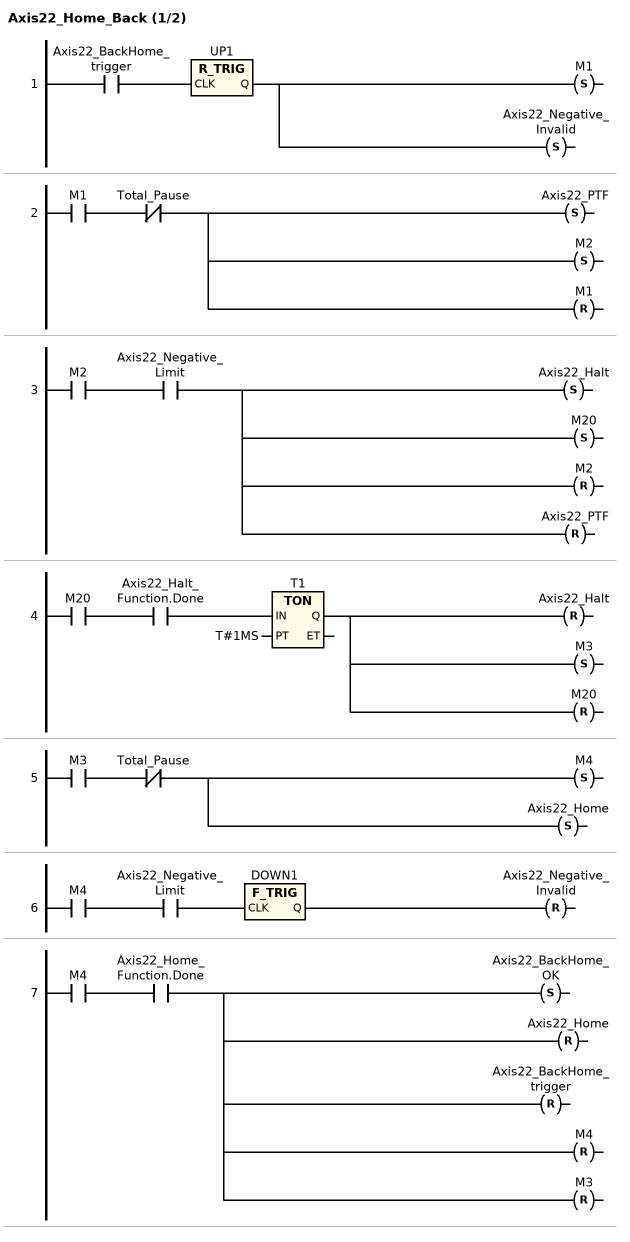
[picture p96: Axis22_Home_Back (LD)]
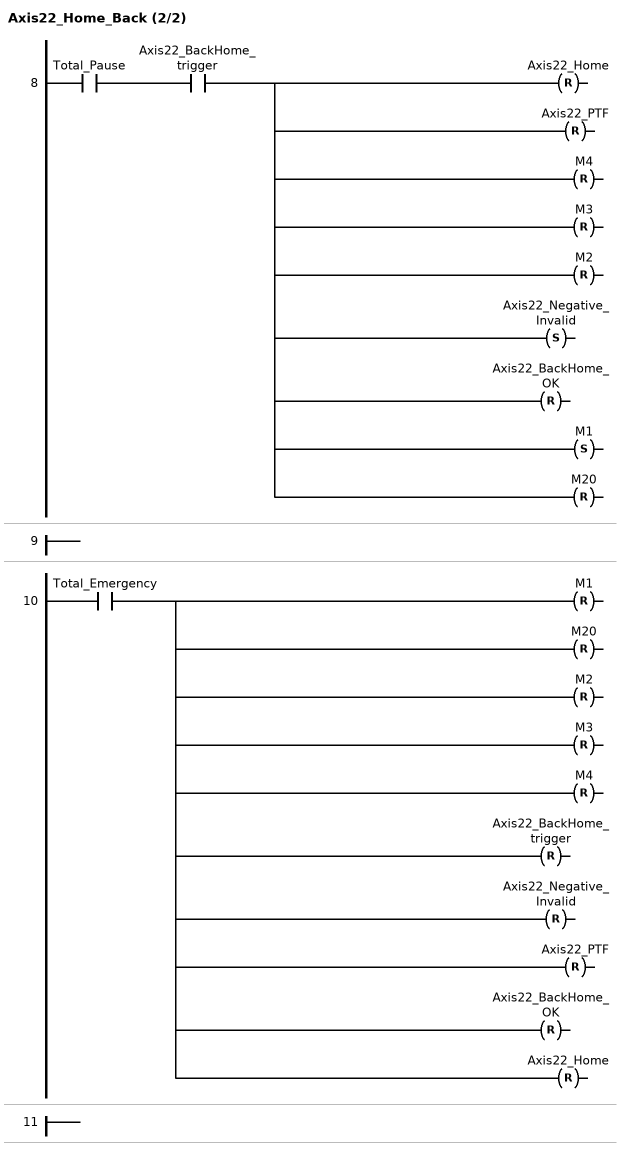
_LD_ (* Ladder Diagram *)
NETWORK 1
	[Axis22_BackHome_trigger] - UP1:R_TRIG(CLK: *) --- (S M1) (S Axis22_Negative_Invalid)
NETWORK 2
	[M1] - [/Total_Pause] --- (S Axis22_PTF) (S M2) (R M1)
NETWORK 3
	[M2] - [Axis22_Negative_Limit] --- (S Axis22_Halt) (S M20) (R M2) (R Axis22_PTF)
NETWORK 4
	[M20] - [Axis22_Halt_Function.Done] - T1:TON(IN: *, PT: T#1MS) --- (R Axis22_Halt) (S M3) (R M20)
NETWORK 5
	[M3] - [/Total_Pause] --- (S M4) (S Axis22_Home)
NETWORK 6
	[M4] - [Axis22_Negative_Limit] - DOWN1:F_TRIG(CLK: *) --- (R Axis22_Negative_Invalid)
NETWORK 7
	[M4] - [Axis22_Home_Function.Done] --- (S Axis22_BackHome_OK) (R Axis22_Home) (R Axis22_BackHome_trigger) (R M4) (R M3)
NETWORK 8
	[Total_Pause] - [Axis22_BackHome_trigger] --- (R Axis22_Home) (R Axis22_PTF) (R M4) (R M3) (R M2) (S Axis22_Negative_Invalid) (R Axis22_BackHome_OK) (S M1) (R M20)
NETWORK 9
	*
NETWORK 10
	[Total_Emergency] --- (R M1) (R M20) (R M2) (R M3) (R M4) (R Axis22_BackHome_trigger) (R Axis22_Negative_Invalid) (R Axis22_PTF) (R Axis22_BackHome_OK) (R Axis22_Home)
NETWORK 11
	*
_END_LD_
(* the same logic as Structured Text *)
(* Network 1 *)
UP1(CLK := Axis22_BackHome_trigger);
IF UP1.Q THEN M1 := TRUE; Axis22_Negative_Invalid := TRUE; END_IF;
(* Network 2 *)
_p1 := M1 AND NOT Total_Pause;
IF _p1 THEN Axis22_PTF := TRUE; M2 := TRUE; M1 := FALSE; END_IF;
(* Network 3 *)
_p2 := M2 AND Axis22_Negative_Limit;
IF _p2 THEN Axis22_Halt := TRUE; M20 := TRUE; M2 := FALSE; Axis22_PTF := FALSE; END_IF;
(* Network 4 *)
T1(IN := M20 AND Axis22_Halt_Function.Done, PT := T#1MS);
IF T1.Q THEN Axis22_Halt := FALSE; M3 := TRUE; M20 := FALSE; END_IF;
(* Network 5 *)
IF M3 AND NOT Total_Pause THEN M4 := TRUE; Axis22_Home := TRUE; END_IF;
(* Network 6 *)
DOWN1(CLK := M4 AND Axis22_Negative_Limit);
IF DOWN1.Q THEN Axis22_Negative_Invalid := FALSE; END_IF;
(* Network 7 *)
_p3 := M4 AND Axis22_Home_Function.Done;
IF _p3 THEN Axis22_BackHome_OK := TRUE; Axis22_Home := FALSE; Axis22_BackHome_trigger := FALSE; M4 := FALSE; M3 := FALSE; END_IF;
(* Network 8 *)
IF Total_Pause AND Axis22_BackHome_trigger THEN Axis22_Home := FALSE; Axis22_PTF := FALSE; M4 := FALSE; M3 := FALSE; M2 := FALSE; Axis22_Negative_Invalid := TRUE; Axis22_BackHome_OK := FALSE; M1 := TRUE; M20 := FALSE; END_IF;
(* Network 9 *)
(* Network 10 *)
IF Total_Emergency THEN M1 := FALSE; M20 := FALSE; M2 := FALSE; M3 := FALSE; M4 := FALSE; Axis22_BackHome_trigger := FALSE; Axis22_Negative_Invalid := FALSE; Axis22_PTF := FALSE; Axis22_BackHome_OK := FALSE; Axis22_Home := FALSE; END_IF;
(* Network 11 *)
END_PROGRAM

(* POU Other_Folder/Home_Back/Axis23_Home_Back, LD *)
PROGRAM Axis23_Home_Back
VAR
	UP1: R_TRIG;
	M1: BOOL;
	M2: BOOL;
	UP2: R_TRIG;
	T1: TON;
	M3: BOOL;
	M4: BOOL;
	DOWN1: F_TRIG;
	M20: BOOL;
END_VAR
VAR (* helpers for the ST form of the networks *)
	_p1 : BOOL;
	_p2 : BOOL;
	_p3 : BOOL;
END_VAR
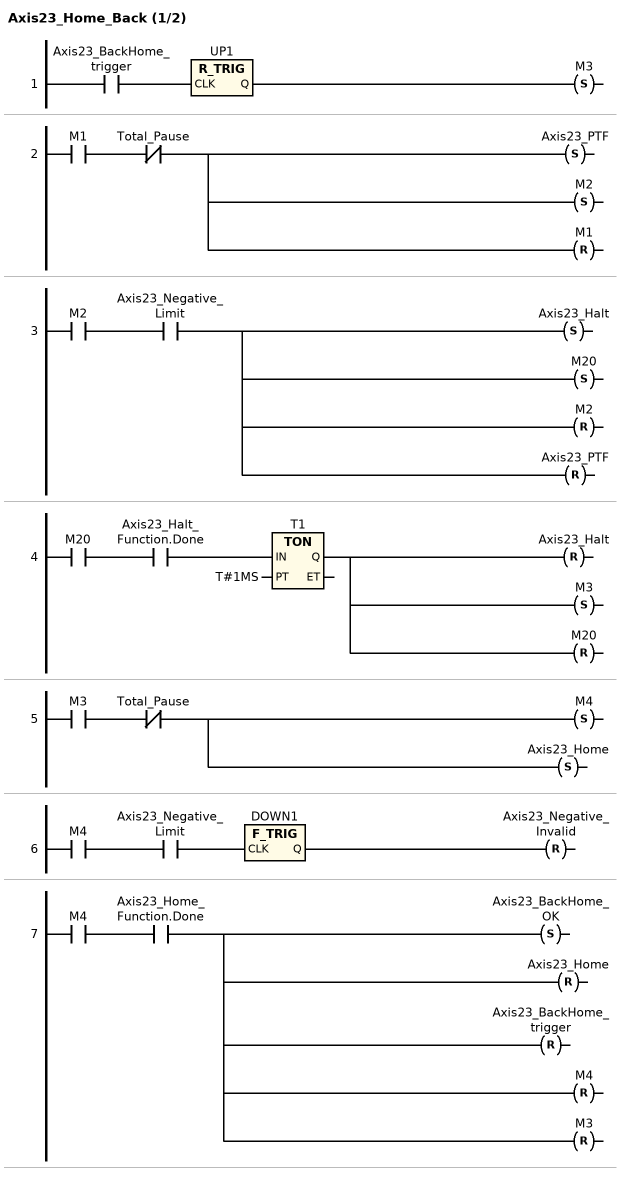
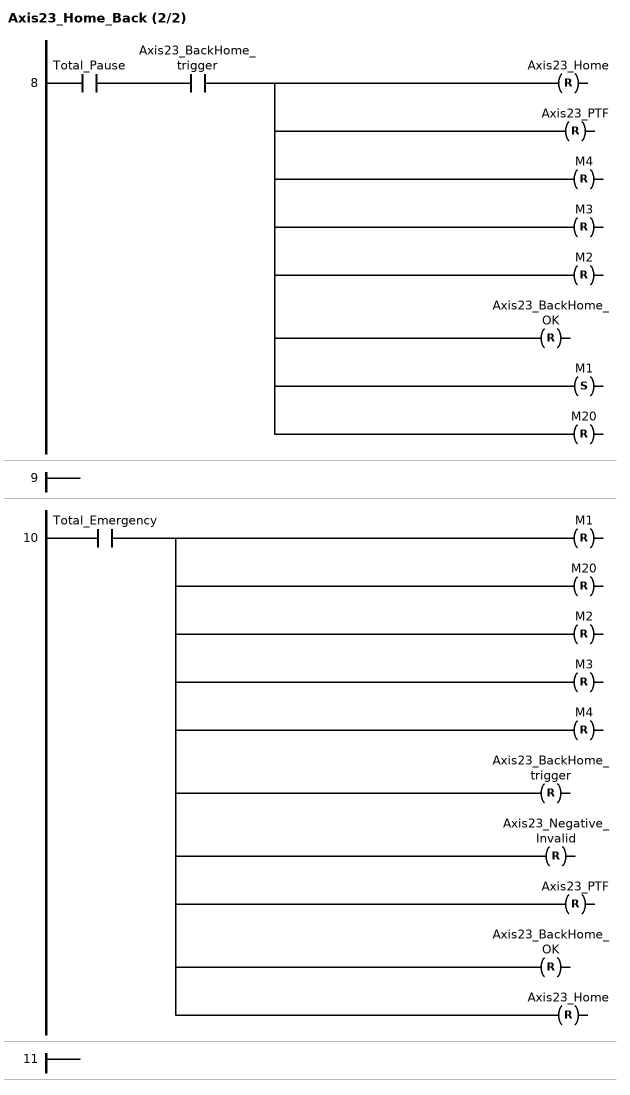
_LD_ (* Ladder Diagram *)
NETWORK 1
	[Axis23_BackHome_trigger] - UP1:R_TRIG(CLK: *) --- (S M3)
NETWORK 2
	[M1] - [/Total_Pause] --- (S Axis23_PTF) (S M2) (R M1)
NETWORK 3
	[M2] - [Axis23_Negative_Limit] --- (S Axis23_Halt) (S M20) (R M2) (R Axis23_PTF)
NETWORK 4
	[M20] - [Axis23_Halt_Function.Done] - T1:TON(IN: *, PT: T#1MS) --- (R Axis23_Halt) (S M3) (R M20)
NETWORK 5
	[M3] - [/Total_Pause] --- (S M4) (S Axis23_Home)
NETWORK 6
	[M4] - [Axis23_Negative_Limit] - DOWN1:F_TRIG(CLK: *) --- (R Axis23_Negative_Invalid)
NETWORK 7
	[M4] - [Axis23_Home_Function.Done] --- (S Axis23_BackHome_OK) (R Axis23_Home) (R Axis23_BackHome_trigger) (R M4) (R M3)
NETWORK 8
	[Total_Pause] - [Axis23_BackHome_trigger] --- (R Axis23_Home) (R Axis23_PTF) (R M4) (R M3) (R M2) (R Axis23_BackHome_OK) (S M1) (R M20)
NETWORK 9
	*
NETWORK 10
	[Total_Emergency] --- (R M1) (R M20) (R M2) (R M3) (R M4) (R Axis23_BackHome_trigger) (R Axis23_Negative_Invalid) (R Axis23_PTF) (R Axis23_BackHome_OK) (R Axis23_Home)
NETWORK 11
	*
_END_LD_
(* the same logic as Structured Text *)
(* Network 1 *)
UP1(CLK := Axis23_BackHome_trigger);
IF UP1.Q THEN M3 := TRUE; END_IF;
(* Network 2 *)
_p1 := M1 AND NOT Total_Pause;
IF _p1 THEN Axis23_PTF := TRUE; M2 := TRUE; M1 := FALSE; END_IF;
(* Network 3 *)
_p2 := M2 AND Axis23_Negative_Limit;
IF _p2 THEN Axis23_Halt := TRUE; M20 := TRUE; M2 := FALSE; Axis23_PTF := FALSE; END_IF;
(* Network 4 *)
T1(IN := M20 AND Axis23_Halt_Function.Done, PT := T#1MS);
IF T1.Q THEN Axis23_Halt := FALSE; M3 := TRUE; M20 := FALSE; END_IF;
(* Network 5 *)
IF M3 AND NOT Total_Pause THEN M4 := TRUE; Axis23_Home := TRUE; END_IF;
(* Network 6 *)
DOWN1(CLK := M4 AND Axis23_Negative_Limit);
IF DOWN1.Q THEN Axis23_Negative_Invalid := FALSE; END_IF;
(* Network 7 *)
_p3 := M4 AND Axis23_Home_Function.Done;
IF _p3 THEN Axis23_BackHome_OK := TRUE; Axis23_Home := FALSE; Axis23_BackHome_trigger := FALSE; M4 := FALSE; M3 := FALSE; END_IF;
(* Network 8 *)
IF Total_Pause AND Axis23_BackHome_trigger THEN Axis23_Home := FALSE; Axis23_PTF := FALSE; M4 := FALSE; M3 := FALSE; M2 := FALSE; Axis23_BackHome_OK := FALSE; M1 := TRUE; M20 := FALSE; END_IF;
(* Network 9 *)
(* Network 10 *)
IF Total_Emergency THEN M1 := FALSE; M20 := FALSE; M2 := FALSE; M3 := FALSE; M4 := FALSE; Axis23_BackHome_trigger := FALSE; Axis23_Negative_Invalid := FALSE; Axis23_PTF := FALSE; Axis23_BackHome_OK := FALSE; Axis23_Home := FALSE; END_IF;
(* Network 11 *)
END_PROGRAM

(* POU Other_Folder/Home_Back/Axis24_Home_Back, LD *)
PROGRAM Axis24_Home_Back
VAR
	UP1: R_TRIG;
	M1: BOOL;
	M2: BOOL;
	UP2: R_TRIG;
	T1: TON;
	M3: BOOL;
	M4: BOOL;
	DOWN1: F_TRIG;
	M20: BOOL;
END_VAR
VAR (* helpers for the ST form of the networks *)
	_p1 : BOOL;
	_p2 : BOOL;
	_p3 : BOOL;
END_VAR
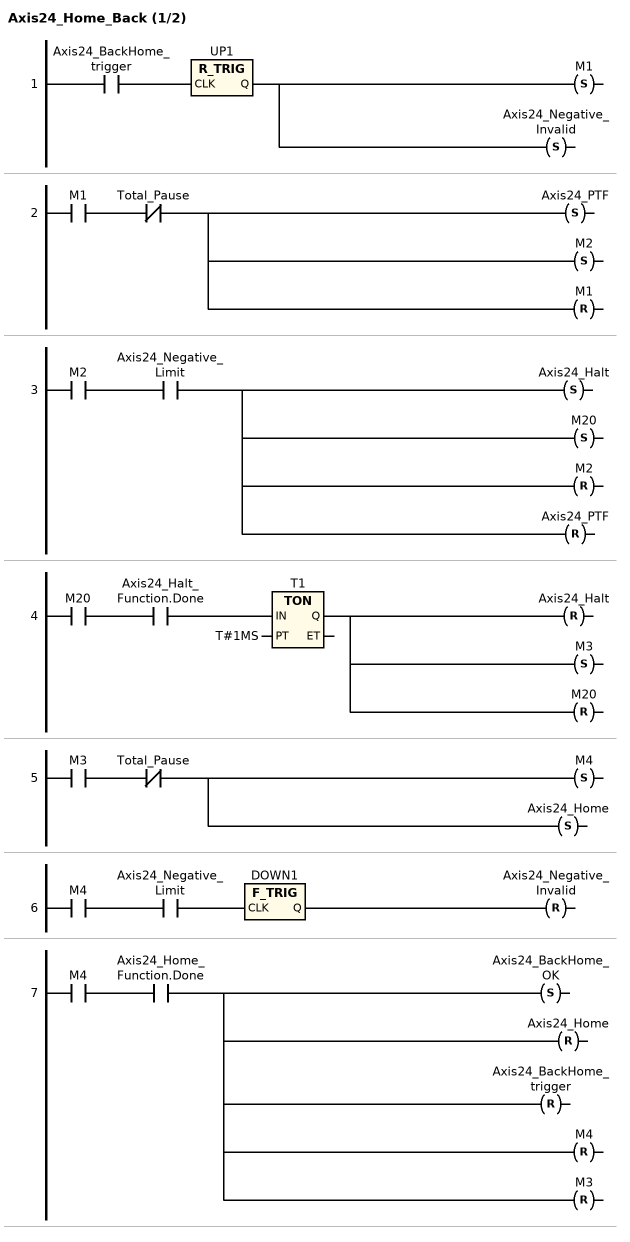
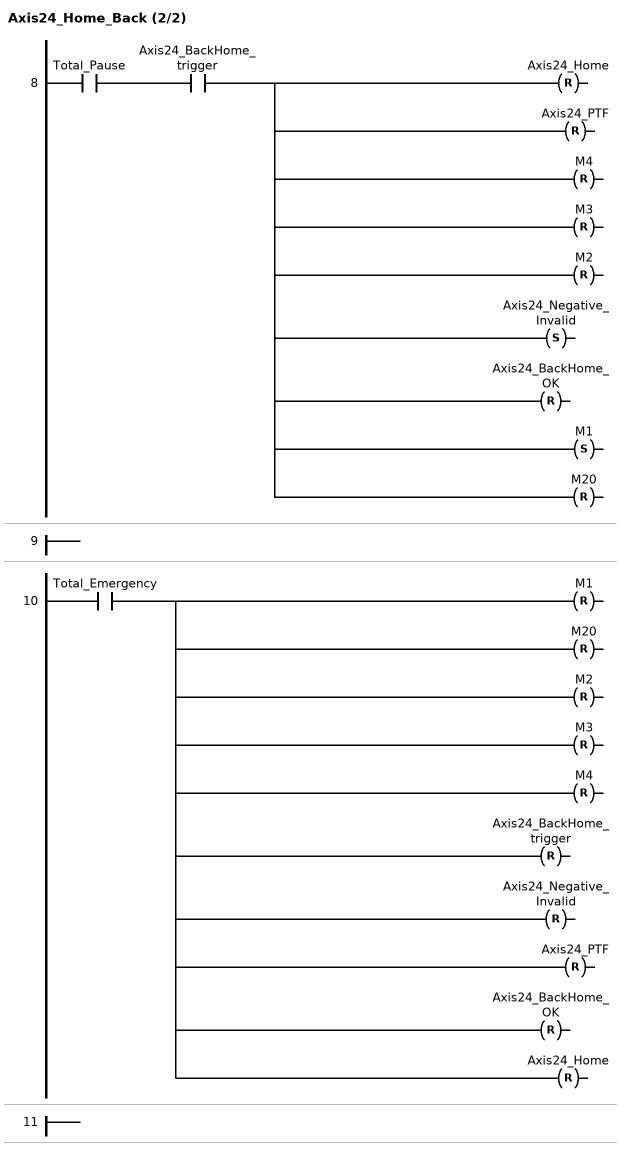
_LD_ (* Ladder Diagram *)
NETWORK 1
	[Axis24_BackHome_trigger] - UP1:R_TRIG(CLK: *) --- (S M1) (S Axis24_Negative_Invalid)
NETWORK 2
	[M1] - [/Total_Pause] --- (S Axis24_PTF) (S M2) (R M1)
NETWORK 3
	[M2] - [Axis24_Negative_Limit] --- (S Axis24_Halt) (S M20) (R M2) (R Axis24_PTF)
NETWORK 4
	[M20] - [Axis24_Halt_Function.Done] - T1:TON(IN: *, PT: T#1MS) --- (R Axis24_Halt) (S M3) (R M20)
NETWORK 5
	[M3] - [/Total_Pause] --- (S M4) (S Axis24_Home)
NETWORK 6
	[M4] - [Axis24_Negative_Limit] - DOWN1:F_TRIG(CLK: *) --- (R Axis24_Negative_Invalid)
NETWORK 7
	[M4] - [Axis24_Home_Function.Done] --- (S Axis24_BackHome_OK) (R Axis24_Home) (R Axis24_BackHome_trigger) (R M4) (R M3)
NETWORK 8
	[Total_Pause] - [Axis24_BackHome_trigger] --- (R Axis24_Home) (R Axis24_PTF) (R M4) (R M3) (R M2) (S Axis24_Negative_Invalid) (R Axis24_BackHome_OK) (S M1) (R M20)
NETWORK 9
	*
NETWORK 10
	[Total_Emergency] --- (R M1) (R M20) (R M2) (R M3) (R M4) (R Axis24_BackHome_trigger) (R Axis24_Negative_Invalid) (R Axis24_PTF) (R Axis24_BackHome_OK) (R Axis24_Home)
NETWORK 11
	*
_END_LD_
(* the same logic as Structured Text *)
(* Network 1 *)
UP1(CLK := Axis24_BackHome_trigger);
IF UP1.Q THEN M1 := TRUE; Axis24_Negative_Invalid := TRUE; END_IF;
(* Network 2 *)
_p1 := M1 AND NOT Total_Pause;
IF _p1 THEN Axis24_PTF := TRUE; M2 := TRUE; M1 := FALSE; END_IF;
(* Network 3 *)
_p2 := M2 AND Axis24_Negative_Limit;
IF _p2 THEN Axis24_Halt := TRUE; M20 := TRUE; M2 := FALSE; Axis24_PTF := FALSE; END_IF;
(* Network 4 *)
T1(IN := M20 AND Axis24_Halt_Function.Done, PT := T#1MS);
IF T1.Q THEN Axis24_Halt := FALSE; M3 := TRUE; M20 := FALSE; END_IF;
(* Network 5 *)
IF M3 AND NOT Total_Pause THEN M4 := TRUE; Axis24_Home := TRUE; END_IF;
(* Network 6 *)
DOWN1(CLK := M4 AND Axis24_Negative_Limit);
IF DOWN1.Q THEN Axis24_Negative_Invalid := FALSE; END_IF;
(* Network 7 *)
_p3 := M4 AND Axis24_Home_Function.Done;
IF _p3 THEN Axis24_BackHome_OK := TRUE; Axis24_Home := FALSE; Axis24_BackHome_trigger := FALSE; M4 := FALSE; M3 := FALSE; END_IF;
(* Network 8 *)
IF Total_Pause AND Axis24_BackHome_trigger THEN Axis24_Home := FALSE; Axis24_PTF := FALSE; M4 := FALSE; M3 := FALSE; M2 := FALSE; Axis24_Negative_Invalid := TRUE; Axis24_BackHome_OK := FALSE; M1 := TRUE; M20 := FALSE; END_IF;
(* Network 9 *)
(* Network 10 *)
IF Total_Emergency THEN M1 := FALSE; M20 := FALSE; M2 := FALSE; M3 := FALSE; M4 := FALSE; Axis24_BackHome_trigger := FALSE; Axis24_Negative_Invalid := FALSE; Axis24_PTF := FALSE; Axis24_BackHome_OK := FALSE; Axis24_Home := FALSE; END_IF;
(* Network 11 *)
END_PROGRAM

(* POU Other_Folder/Home_Back/Axis25_Home_Back, LD *)
PROGRAM Axis25_Home_Back
VAR
	UP1: R_TRIG;
	M1: BOOL;
	M2: BOOL;
	UP2: R_TRIG;
	T1: TON;
	T2: TON;
	M3: BOOL;
	M4: BOOL;
	DOWN1: F_TRIG;
	M20: BOOL;
END_VAR
VAR (* helpers for the ST form of the networks *)
	_p1 : BOOL;
	_p2 : BOOL;
END_VAR
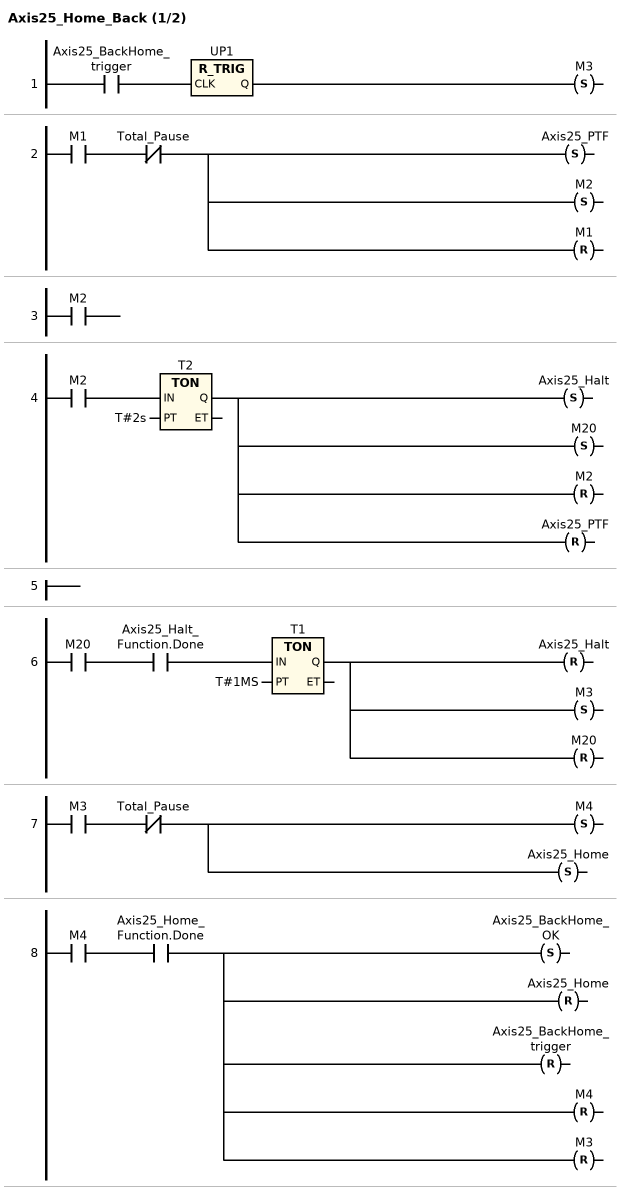
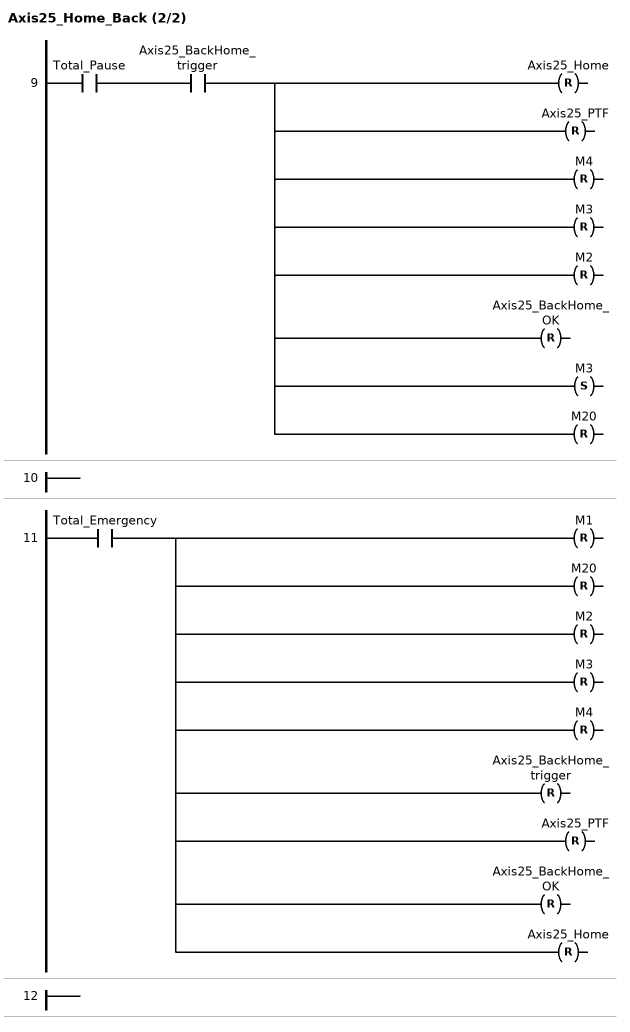
_LD_ (* Ladder Diagram *)
NETWORK 1
	[Axis25_BackHome_trigger] - UP1:R_TRIG(CLK: *) --- (S M3)
NETWORK 2
	[M1] - [/Total_Pause] --- (S Axis25_PTF) (S M2) (R M1)
NETWORK 3
	[M2]
NETWORK 4
	[M2] - T2:TON(IN: *, PT: T#2s) --- (S Axis25_Halt) (S M20) (R M2) (R Axis25_PTF)
NETWORK 5
	*
NETWORK 6
	[M20] - [Axis25_Halt_Function.Done] - T1:TON(IN: *, PT: T#1MS) --- (R Axis25_Halt) (S M3) (R M20)
NETWORK 7
	[M3] - [/Total_Pause] --- (S M4) (S Axis25_Home)
NETWORK 8
	[M4] - [Axis25_Home_Function.Done] --- (S Axis25_BackHome_OK) (R Axis25_Home) (R Axis25_BackHome_trigger) (R M4) (R M3)
NETWORK 9
	[Total_Pause] - [Axis25_BackHome_trigger] --- (R Axis25_Home) (R Axis25_PTF) (R M4) (R M3) (R M2) (R Axis25_BackHome_OK) (S M3) (R M20)
NETWORK 10
	*
NETWORK 11
	[Total_Emergency] --- (R M1) (R M20) (R M2) (R M3) (R M4) (R Axis25_BackHome_trigger) (R Axis25_PTF) (R Axis25_BackHome_OK) (R Axis25_Home)
NETWORK 12
	*
_END_LD_
(* the same logic as Structured Text *)
(* Network 1 *)
UP1(CLK := Axis25_BackHome_trigger);
IF UP1.Q THEN M3 := TRUE; END_IF;
(* Network 2 *)
_p1 := M1 AND NOT Total_Pause;
IF _p1 THEN Axis25_PTF := TRUE; M2 := TRUE; M1 := FALSE; END_IF;
(* Network 3 *)
(* Network 4 *)
T2(IN := M2, PT := T#2s);
IF T2.Q THEN Axis25_Halt := TRUE; M20 := TRUE; M2 := FALSE; Axis25_PTF := FALSE; END_IF;
(* Network 5 *)
(* Network 6 *)
T1(IN := M20 AND Axis25_Halt_Function.Done, PT := T#1MS);
IF T1.Q THEN Axis25_Halt := FALSE; M3 := TRUE; M20 := FALSE; END_IF;
(* Network 7 *)
IF M3 AND NOT Total_Pause THEN M4 := TRUE; Axis25_Home := TRUE; END_IF;
(* Network 8 *)
_p2 := M4 AND Axis25_Home_Function.Done;
IF _p2 THEN Axis25_BackHome_OK := TRUE; Axis25_Home := FALSE; Axis25_BackHome_trigger := FALSE; M4 := FALSE; M3 := FALSE; END_IF;
(* Network 9 *)
IF Total_Pause AND Axis25_BackHome_trigger THEN Axis25_Home := FALSE; Axis25_PTF := FALSE; M4 := FALSE; M3 := FALSE; M2 := FALSE; Axis25_BackHome_OK := FALSE; M3 := TRUE; M20 := FALSE; END_IF;
(* Network 10 *)
(* Network 11 *)
IF Total_Emergency THEN M1 := FALSE; M20 := FALSE; M2 := FALSE; M3 := FALSE; M4 := FALSE; Axis25_BackHome_trigger := FALSE; Axis25_PTF := FALSE; Axis25_BackHome_OK := FALSE; Axis25_Home := FALSE; END_IF;
(* Network 12 *)
END_PROGRAM

(* POU Other_Folder/Home_Back/Home_Ptf_Rst, ST *)
PROGRAM Home_Ptf_Rst
VAR
END_VAR
IF Total_Pause OR Total_Emergency THEN
	Axis1_Home:=FALSE;
	Axis2_Home:=FALSE;
	Axis3_Home:=FALSE;
	Axis4_Home:=FALSE;
	Axis5_Home:=FALSE;
	Axis6_Home:=FALSE;
	Axis7_Home:=FALSE;
	Axis8_Home:=FALSE;
	Axis9_Home:=FALSE;
	Axis10_Home:=FALSE;
	Axis11_Home:=FALSE;
	Axis21_Home:=FALSE;
	Axis22_Home:=FALSE;
	Axis23_Home:=FALSE;
	Axis24_Home:=FALSE;
	Axis25_Home:=FALSE;

	Axis1_MoveAbsolute:=FALSE;
	Axis2_MoveAbsolute:=FALSE;
	Axis3_MoveAbsolute:=FALSE;
	Axis4_MoveAbsolute:=FALSE;
	Axis5_MoveAbsolute:=FALSE;
	Axis4_1_MoveAbsolute:=FALSE;
	Axis5_1_MoveAbsolute:=FALSE;
	Axis6_MoveAbsolute:=FALSE;
	Axis7_MoveAbsolute:=FALSE;
	Axis8_MoveAbsolute:=FALSE;
	Axis9_MoveAbsolute:=FALSE;
	Axis10_MoveAbsolute:=FALSE;
	Axis10_MoveAbsolute1:=FALSE;
	Axis11_MoveAbsolute:=FALSE;
	Axis21_MoveAbsolute:=FALSE;
	Axis22_MoveAbsolute:=FALSE;
	Axis23_MoveAbsolute:=FALSE;
	Axis24_MoveAbsolute:=FALSE;
	Axis25_MoveAbsolute:=FALSE;


	Axis1_PTF:=FALSE;
	Axis2_PTF:=FALSE;
	Axis3_PTF:=FALSE;
	Axis4_PTF:=FALSE;
	Axis5_PTF:=FALSE;
	Axis6_PTF:=FALSE;
	Axis7_PTF:=FALSE;
	Axis8_PTF:=FALSE;
	Axis9_PTF:=FALSE;
	Axis10_PTF:=FALSE;
	Axis11_PTF:=FALSE;
	Axis3_PTF_2:=FALSE;
	Axis6_PTF_2:=FALSE;
	Axis7_PTF_2:=FALSE;
	Axis8_PTF_2:=FALSE;
	Axis9_PTF_2:=FALSE;
	Axis21_PTF:=FALSE;
	Axis22_PTF:=FALSE;
	Axis23_PTF:=FALSE;
	Axis24_PTF:=FALSE;
	Axis25_PTF:=FALSE;
END_IF
END_PROGRAM

(* POU Other_Folder/Akam_Stop_Message/Alarm_Monitoring, LD *)
PROGRAM Alarm_Monitoring
VAR
	T1: TON;
	T2: TON;
	T3: TON;
	T4: TON;
	T5: TON;
	T6: TON;
	T7: TON;
	T8: TON;
	T100: TON;
	T101: TON;

	M99: BOOL;

	UP2: R_TRIG;

END_VAR
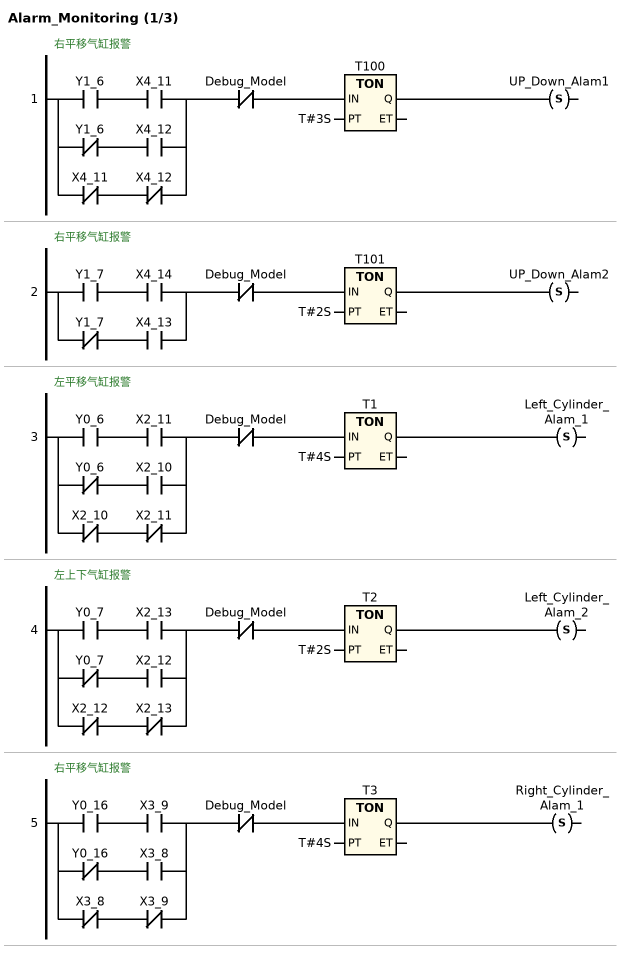
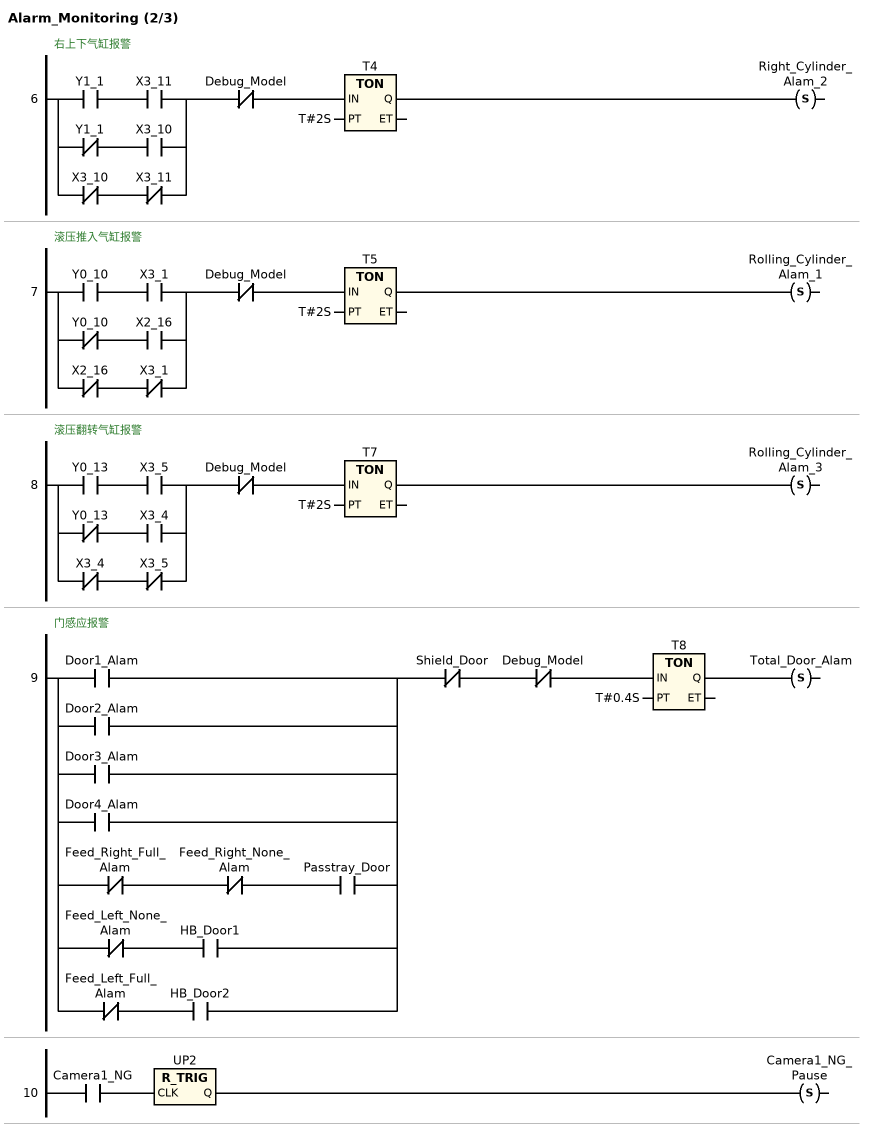
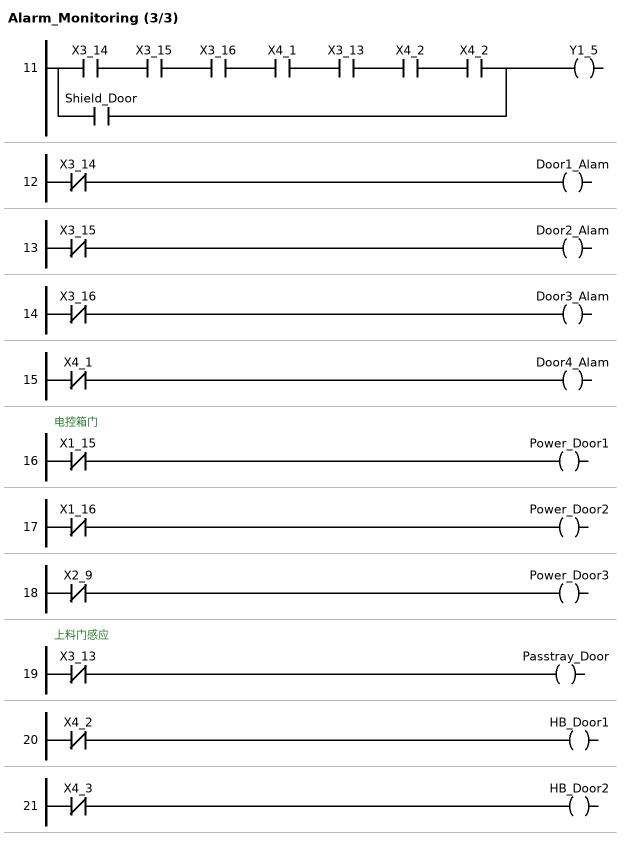
_LD_ (* Ladder Diagram *)
NETWORK 1 (* 右平移气缸报警 *)
	{ [Y1_6] - [X4_11] | [/Y1_6] - [X4_12] | [/X4_11] - [/X4_12] } - [/Debug_Model] - T100:TON(IN: *, PT: T#3S) --- (S UP_Down_Alam1)
NETWORK 2 (* 右平移气缸报警 *)
	{ [Y1_7] - [X4_14] | [/Y1_7] - [X4_13] } - [/Debug_Model] - T101:TON(IN: *, PT: T#2S) --- (S UP_Down_Alam2)
NETWORK 3 (* 左平移气缸报警 *)
	{ [Y0_6] - [X2_11] | [/Y0_6] - [X2_10] | [/X2_10] - [/X2_11] } - [/Debug_Model] - T1:TON(IN: *, PT: T#4S) --- (S Left_Cylinder_Alam_1)
NETWORK 4 (* 左上下气缸报警 *)
	{ [Y0_7] - [X2_13] | [/Y0_7] - [X2_12] | [/X2_12] - [/X2_13] } - [/Debug_Model] - T2:TON(IN: *, PT: T#2S) --- (S Left_Cylinder_Alam_2)
NETWORK 5 (* 右平移气缸报警 *)
	{ [Y0_16] - [X3_9] | [/Y0_16] - [X3_8] | [/X3_8] - [/X3_9] } - [/Debug_Model] - T3:TON(IN: *, PT: T#4S) --- (S Right_Cylinder_Alam_1)
NETWORK 6 (* 右上下气缸报警 *)
	{ [Y1_1] - [X3_11] | [/Y1_1] - [X3_10] | [/X3_10] - [/X3_11] } - [/Debug_Model] - T4:TON(IN: *, PT: T#2S) --- (S Right_Cylinder_Alam_2)
NETWORK 7 (* 滚压推入气缸报警 *)
	{ [Y0_10] - [X3_1] | [/Y0_10] - [X2_16] | [/X2_16] - [/X3_1] } - [/Debug_Model] - T5:TON(IN: *, PT: T#2S) --- (S Rolling_Cylinder_Alam_1)
NETWORK 8 (* 滚压翻转气缸报警 *)
	{ [Y0_13] - [X3_5] | [/Y0_13] - [X3_4] | [/X3_4] - [/X3_5] } - [/Debug_Model] - T7:TON(IN: *, PT: T#2S) --- (S Rolling_Cylinder_Alam_3)
NETWORK 9 (* 门感应报警 *)
	{ [Door1_Alam] | [Door2_Alam] | [Door3_Alam] | [Door4_Alam] | [/Feed_Right_Full_Alam] - [/Feed_Right_None_Alam] - [Passtray_Door] | [/Feed_Left_None_Alam] - [HB_Door1] | [/Feed_Left_Full_Alam] - [HB_Door2] } - [/Shield_Door] - [/Debug_Model] - T8:TON(IN: *, PT: T#0.4S) --- (S Total_Door_Alam)
NETWORK 10
	[Camera1_NG] - UP2:R_TRIG(CLK: *) --- (S Camera1_NG_Pause)
NETWORK 11
	{ [X3_14] - [X3_15] - [X3_16] - [X4_1] - [X3_13] - [X4_2] - [X4_2] | [Shield_Door] } --- (Y1_5)
NETWORK 12
	[/X3_14] --- (Door1_Alam)
NETWORK 13
	[/X3_15] --- (Door2_Alam)
NETWORK 14
	[/X3_16] --- (Door3_Alam)
NETWORK 15
	[/X4_1] --- (Door4_Alam)
NETWORK 16 (* 电控箱门 *)
	[/X1_15] --- (Power_Door1)
NETWORK 17
	[/X1_16] --- (Power_Door2)
NETWORK 18
	[/X2_9] --- (Power_Door3)
NETWORK 19 (* 上料门感应 *)
	[/X3_13] --- (Passtray_Door)
NETWORK 20
	[/X4_2] --- (HB_Door1)
NETWORK 21
	[/X4_3] --- (HB_Door2)
_END_LD_
(* the same logic as Structured Text *)
(* Network 1: 右平移气缸报警 *)
T100(IN := (Y1_6 AND X4_11 OR NOT Y1_6 AND X4_12 OR NOT X4_11 AND NOT X4_12) AND NOT Debug_Model, PT := T#3S);
IF T100.Q THEN UP_Down_Alam1 := TRUE; END_IF;
(* Network 2: 右平移气缸报警 *)
T101(IN := (Y1_7 AND X4_14 OR NOT Y1_7 AND X4_13) AND NOT Debug_Model, PT := T#2S);
IF T101.Q THEN UP_Down_Alam2 := TRUE; END_IF;
(* Network 3: 左平移气缸报警 *)
T1(IN := (Y0_6 AND X2_11 OR NOT Y0_6 AND X2_10 OR NOT X2_10 AND NOT X2_11) AND NOT Debug_Model, PT := T#4S);
IF T1.Q THEN Left_Cylinder_Alam_1 := TRUE; END_IF;
(* Network 4: 左上下气缸报警 *)
T2(IN := (Y0_7 AND X2_13 OR NOT Y0_7 AND X2_12 OR NOT X2_12 AND NOT X2_13) AND NOT Debug_Model, PT := T#2S);
IF T2.Q THEN Left_Cylinder_Alam_2 := TRUE; END_IF;
(* Network 5: 右平移气缸报警 *)
T3(IN := (Y0_16 AND X3_9 OR NOT Y0_16 AND X3_8 OR NOT X3_8 AND NOT X3_9) AND NOT Debug_Model, PT := T#4S);
IF T3.Q THEN Right_Cylinder_Alam_1 := TRUE; END_IF;
(* Network 6: 右上下气缸报警 *)
T4(IN := (Y1_1 AND X3_11 OR NOT Y1_1 AND X3_10 OR NOT X3_10 AND NOT X3_11) AND NOT Debug_Model, PT := T#2S);
IF T4.Q THEN Right_Cylinder_Alam_2 := TRUE; END_IF;
(* Network 7: 滚压推入气缸报警 *)
T5(IN := (Y0_10 AND X3_1 OR NOT Y0_10 AND X2_16 OR NOT X2_16 AND NOT X3_1) AND NOT Debug_Model, PT := T#2S);
IF T5.Q THEN Rolling_Cylinder_Alam_1 := TRUE; END_IF;
(* Network 8: 滚压翻转气缸报警 *)
T7(IN := (Y0_13 AND X3_5 OR NOT Y0_13 AND X3_4 OR NOT X3_4 AND NOT X3_5) AND NOT Debug_Model, PT := T#2S);
IF T7.Q THEN Rolling_Cylinder_Alam_3 := TRUE; END_IF;
(* Network 9: 门感应报警 *)
T8(IN := (Door1_Alam OR Door2_Alam OR Door3_Alam OR Door4_Alam OR NOT Feed_Right_Full_Alam AND NOT Feed_Right_None_Alam AND Passtray_Door OR NOT Feed_Left_None_Alam AND HB_Door1 OR NOT Feed_Left_Full_Alam AND HB_Door2) AND NOT Shield_Door AND NOT Debug_Model, PT := T#0.4S);
IF T8.Q THEN Total_Door_Alam := TRUE; END_IF;
(* Network 10 *)
UP2(CLK := Camera1_NG);
IF UP2.Q THEN Camera1_NG_Pause := TRUE; END_IF;
(* Network 11 *)
Y1_5 := X3_14 AND X3_15 AND X3_16 AND X4_1 AND X3_13 AND X4_2 AND X4_2 OR Shield_Door;
(* Network 12 *)
Door1_Alam := NOT X3_14;
(* Network 13 *)
Door2_Alam := NOT X3_15;
(* Network 14 *)
Door3_Alam := NOT X3_16;
(* Network 15 *)
Door4_Alam := NOT X4_1;
(* Network 16: 电控箱门 *)
Power_Door1 := NOT X1_15;
(* Network 17 *)
Power_Door2 := NOT X1_16;
(* Network 18 *)
Power_Door3 := NOT X2_9;
(* Network 19: 上料门感应 *)
Passtray_Door := NOT X3_13;
(* Network 20 *)
HB_Door1 := NOT X4_2;
(* Network 21 *)
HB_Door2 := NOT X4_3;
END_PROGRAM

(* POU Other_Folder/Akam_Stop_Message/Message_And_Status, ST *)
PROGRAM Message_And_Status
VAR

END_VAR
Message[0]:=Need_Ini;
Message[1]:=IsIniing;
Message[2]:=Model_Choose;
Message[3]:=home_backing;
Message[4]:=Debug_Model;
Message[5]:=runing;

Alam[0]:=Total_Axis_Error;
Alam[1]:=Axis1_Error;
Alam[2]:=Axis2_Error;
Alam[3]:=Axis3_Error;
Alam[4]:=Axis4_Error;
Alam[5]:=Axis5_Error;
Alam[6]:=Axis6_Error;
Alam[7]:=Axis7_Error;
Alam[8]:=Axis8_Error;
Alam[9]:=Axis9_Error;
Alam[10]:=Axis10_Error;
Alam[11]:=Axis11_Error;
Alam[12]:=Total_Emergency;
Alam[13]:=Axis1_Limit_Emergency;
Alam[14]:=Axis2_Limit_Emergency;
Alam[15]:=Axis3_Limit_Emergency;
Alam[16]:=Axis4_Limit_Emergency;
Alam[17]:=Axis5_Limit_Emergency;
Alam[18]:=Axis6_Limit_Emergency;
Alam[19]:=Axis7_Limit_Emergency;
Alam[20]:=Axis8_Limit_Emergency;
Alam[21]:=Axis9_Limit_Emergency;
Alam[22]:=Axis10_Limit_Emergency;
Alam[23]:=Axis11_Limit_Emergency;
Alam[24]:=Total_Pause;
Alam[25]:=Pressure_Fail_1;
Alam[26]:=Pressure_Fail_2;
Alam[27]:=Left_Cylinder_Alam_1;
Alam[28]:=Left_Cylinder_Alam_2;
Alam[29]:=Pressure_Left_Fail;
Alam[30]:=Right_Cylinder_Alam_1;
Alam[31]:=Right_Cylinder_Alam_2;
Alam[32]:=Pressure_Right_Fail;
Alam[33]:=Rolling_Cylinder_Alam_1;
Alam[34]:=Rolling_Cylinder_Alam_2;
Alam[35]:=Rolling_Cylinder_Alam_3;
Alam[36]:=Rolling_Pressure_Fail;
Alam[37]:=UP_Down_Alam1;
Alam[38]:=UP_Down_Alam2;
Alam[39]:=Feed_1_Nome_Alam;
Alam[40]:=Feed_Left_None_Alam;
Alam[41]:=Feed_Left_Full_Alam;
Alam[42]:=Feed_Right_None_Alam;
Alam[43]:=Feed_Right_Full_Alam;
Alam[44]:=Total_Door_Alam;
Alam[45]:=Door1_Alam;
Alam[46]:=Door2_Alam;
Alam[47]:=Door3_Alam;
Alam[48]:=Door4_Alam;
Alam[49]:=Passtray_Door;
Alam[50]:=HB_Door1;
Alam[51]:=HB_Door2;
Alam[52]:=Camera1_NG_Pause;
Alam[53]:=Camera2_NG;
Alam[54]:=Feed1_UnReady;
Alam[55]:=FPC_up_Unready;
Alam[56]:=FPC_down_Unready;
Alam[57]:=TRAY_up_Unready;
Alam[58]:=TRAY_down_Unready;
END_PROGRAM

(* POU Other_Folder/Akam_Stop_Message/Pause, LD *)
PROGRAM Pause
VAR

	ssss: BOOL;
	UPA: R_TRIG;
	UPB: R_TRIG;
END_VAR
VAR (* helpers for the ST form of the networks *)
	_p1 : BOOL;
END_VAR
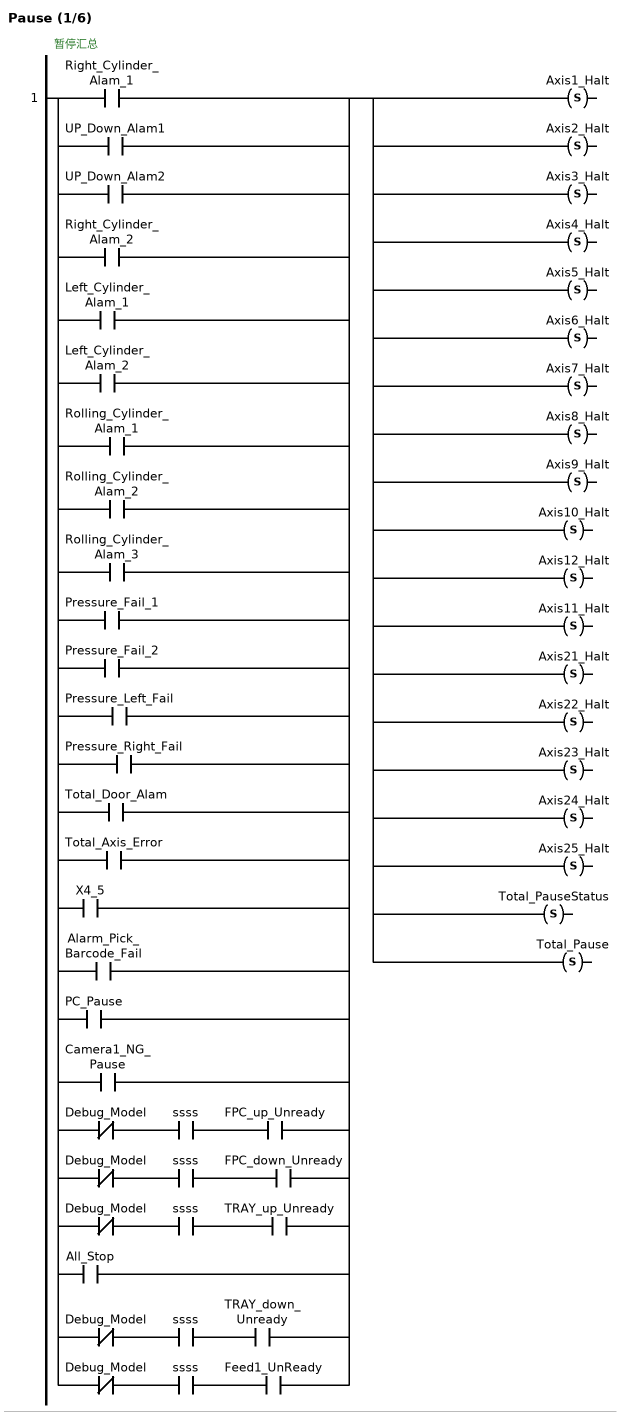
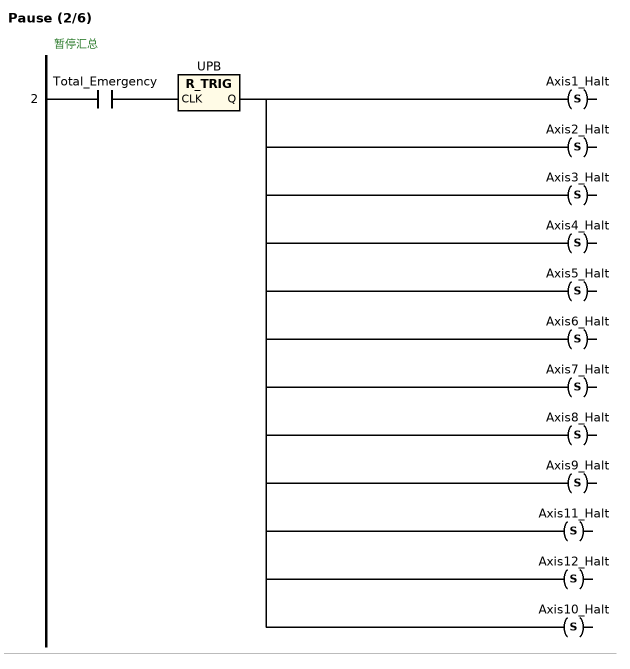
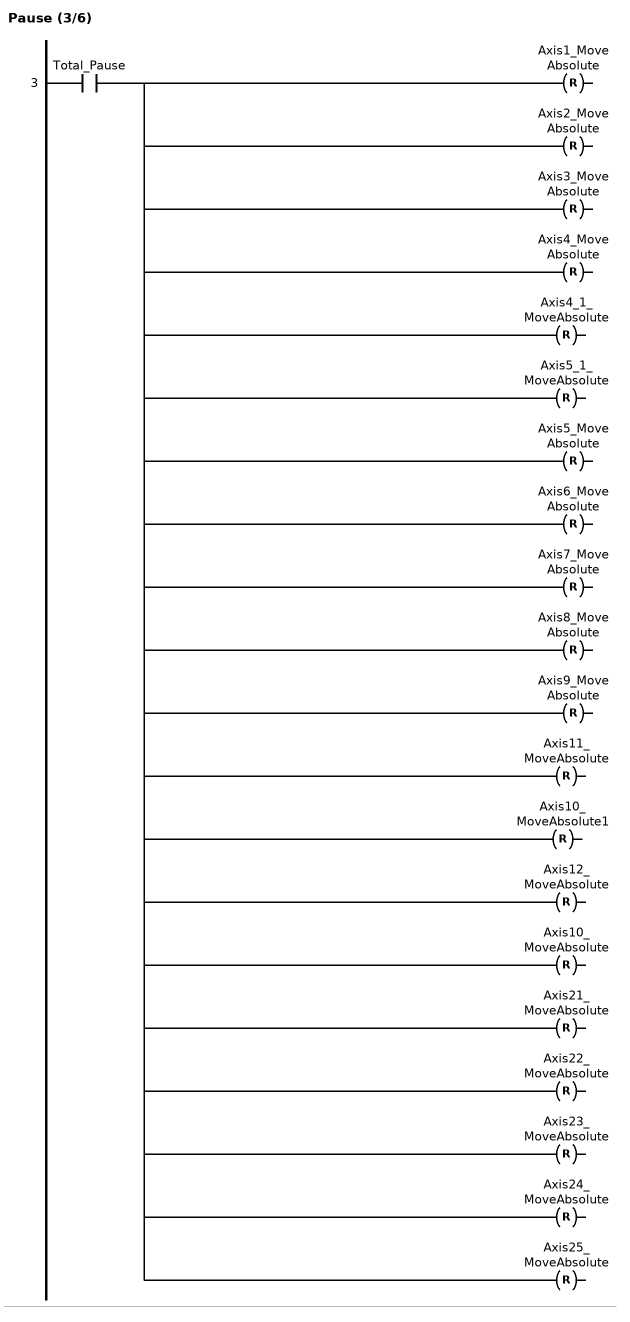
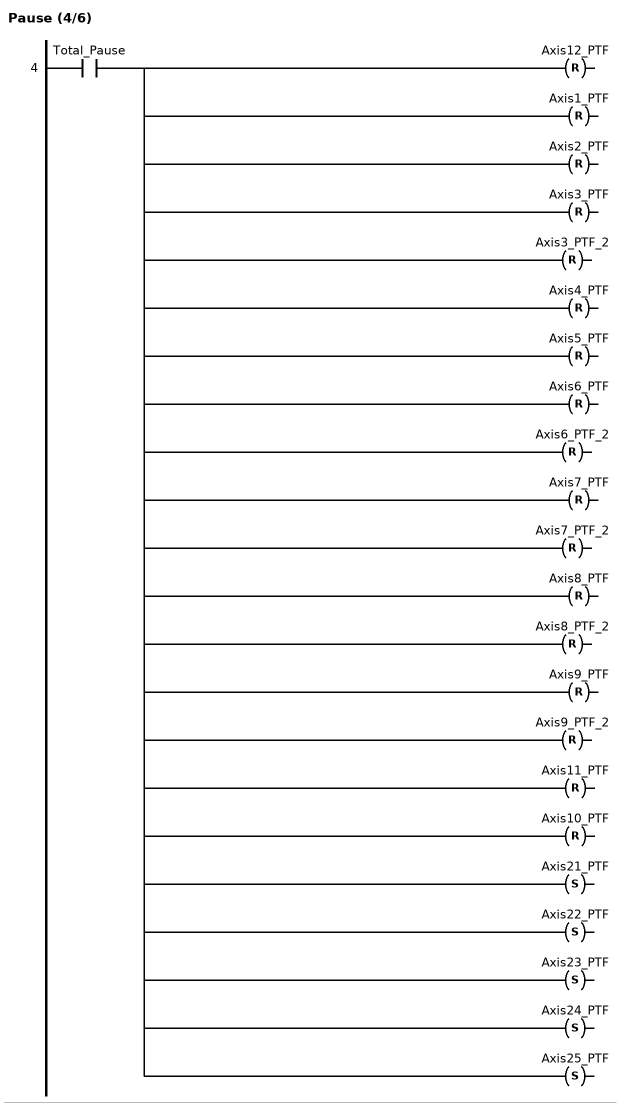
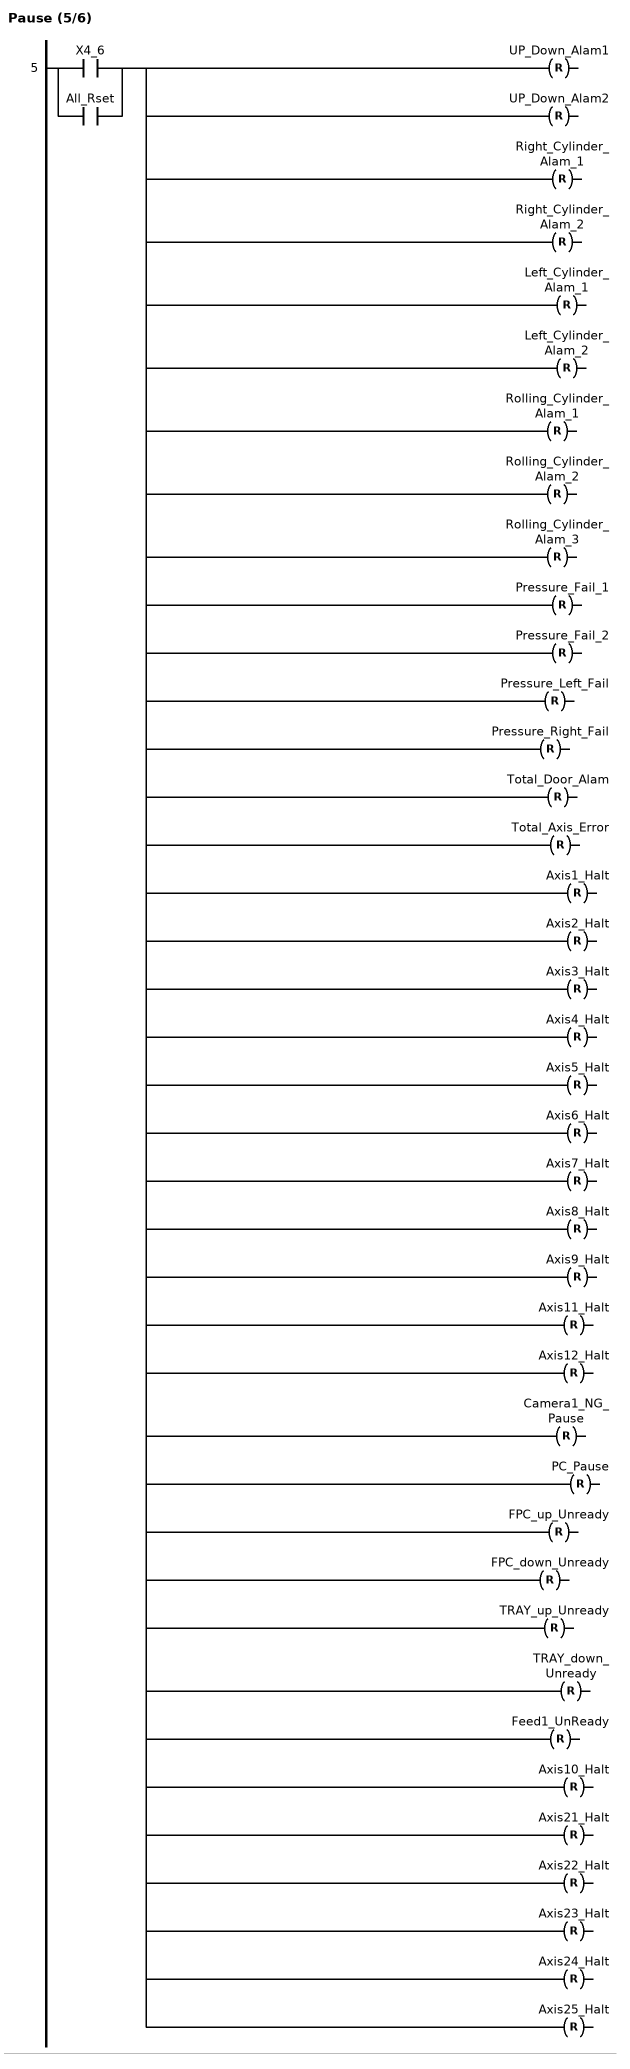
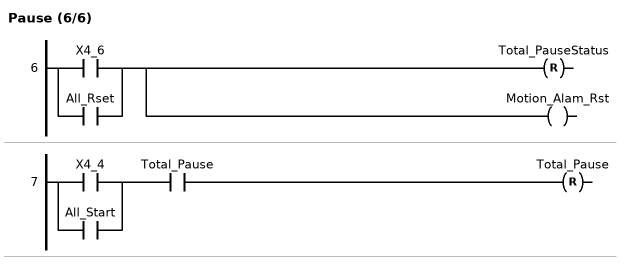
_LD_ (* Ladder Diagram *)
NETWORK 1 (* 暂停汇总 *)
	{ [Right_Cylinder_Alam_1] | [UP_Down_Alam1] | [UP_Down_Alam2] | [Right_Cylinder_Alam_2] | [Left_Cylinder_Alam_1] | [Left_Cylinder_Alam_2] | [Rolling_Cylinder_Alam_1] | [Rolling_Cylinder_Alam_2] | [Rolling_Cylinder_Alam_3] | [Pressure_Fail_1] | [Pressure_Fail_2] | [Pressure_Left_Fail] | [Pressure_Right_Fail] | [Total_Door_Alam] | [Total_Axis_Error] | [X4_5] | [Alarm_Pick_Barcode_Fail] | [PC_Pause] | [Camera1_NG_Pause] | [/Debug_Model] - [ssss] - [FPC_up_Unready] | [/Debug_Model] - [ssss] - [FPC_down_Unready] | [/Debug_Model] - [ssss] - [TRAY_up_Unready] | [All_Stop] | [/Debug_Model] - [ssss] - [TRAY_down_Unready] | [/Debug_Model] - [ssss] - [Feed1_UnReady] } --- (S Axis1_Halt) (S Axis2_Halt) (S Axis3_Halt) (S Axis4_Halt) (S Axis5_Halt) (S Axis6_Halt) (S Axis7_Halt) (S Axis8_Halt) (S Axis9_Halt) (S Axis10_Halt) (S Axis12_Halt) (S Axis11_Halt) (S Axis21_Halt) (S Axis22_Halt) (S Axis23_Halt) (S Axis24_Halt) (S Axis25_Halt) (S Total_PauseStatus) (S Total_Pause)
NETWORK 2 (* 暂停汇总 *)
	[Total_Emergency] - UPB:R_TRIG(CLK: *) --- (S Axis1_Halt) (S Axis2_Halt) (S Axis3_Halt) (S Axis4_Halt) (S Axis5_Halt) (S Axis6_Halt) (S Axis7_Halt) (S Axis8_Halt) (S Axis9_Halt) (S Axis11_Halt) (S Axis12_Halt) (S Axis10_Halt)
NETWORK 3
	[Total_Pause] --- (R Axis1_MoveAbsolute) (R Axis2_MoveAbsolute) (R Axis3_MoveAbsolute) (R Axis4_MoveAbsolute) (R Axis4_1_MoveAbsolute) (R Axis5_1_MoveAbsolute) (R Axis5_MoveAbsolute) (R Axis6_MoveAbsolute) (R Axis7_MoveAbsolute) (R Axis8_MoveAbsolute) (R Axis9_MoveAbsolute) (R Axis11_MoveAbsolute) (R Axis10_MoveAbsolute1) (R Axis12_MoveAbsolute) (R Axis10_MoveAbsolute) (R Axis21_MoveAbsolute) (R Axis22_MoveAbsolute) (R Axis23_MoveAbsolute) (R Axis24_MoveAbsolute) (R Axis25_MoveAbsolute)
NETWORK 4
	[Total_Pause] --- (R Axis12_PTF) (R Axis1_PTF) (R Axis2_PTF) (R Axis3_PTF) (R Axis3_PTF_2) (R Axis4_PTF) (R Axis5_PTF) (R Axis6_PTF) (R Axis6_PTF_2) (R Axis7_PTF) (R Axis7_PTF_2) (R Axis8_PTF) (R Axis8_PTF_2) (R Axis9_PTF) (R Axis9_PTF_2) (R Axis11_PTF) (R Axis10_PTF) (S Axis21_PTF) (S Axis22_PTF) (S Axis23_PTF) (S Axis24_PTF) (S Axis25_PTF)
NETWORK 5
	{ [X4_6] | [All_Rset] } --- (R UP_Down_Alam1) (R UP_Down_Alam2) (R Right_Cylinder_Alam_1) (R Right_Cylinder_Alam_2) (R Left_Cylinder_Alam_1) (R Left_Cylinder_Alam_2) (R Rolling_Cylinder_Alam_1) (R Rolling_Cylinder_Alam_2) (R Rolling_Cylinder_Alam_3) (R Pressure_Fail_1) (R Pressure_Fail_2) (R Pressure_Left_Fail) (R Pressure_Right_Fail) (R Total_Door_Alam) (R Total_Axis_Error) (R Axis1_Halt) (R Axis2_Halt) (R Axis3_Halt) (R Axis4_Halt) (R Axis5_Halt) (R Axis6_Halt) (R Axis7_Halt) (R Axis8_Halt) (R Axis9_Halt) (R Axis11_Halt) (R Axis12_Halt) (R Camera1_NG_Pause) (R PC_Pause) (R FPC_up_Unready) (R FPC_down_Unready) (R TRAY_up_Unready) (R TRAY_down_Unready) (R Feed1_UnReady) (R Axis10_Halt) (R Axis21_Halt) (R Axis22_Halt) (R Axis23_Halt) (R Axis24_Halt) (R Axis25_Halt)
NETWORK 6
	{ [X4_6] | [All_Rset] } --- (R Total_PauseStatus) (Motion_Alam_Rst)
NETWORK 7
	{ [X4_4] | [All_Start] } - [Total_Pause] --- (R Total_Pause)
_END_LD_
(* the same logic as Structured Text *)
(* Network 1: 暂停汇总 *)
_p1 := Right_Cylinder_Alam_1 OR UP_Down_Alam1 OR UP_Down_Alam2 OR Right_Cylinder_Alam_2 OR Left_Cylinder_Alam_1 OR Left_Cylinder_Alam_2 OR Rolling_Cylinder_Alam_1 OR Rolling_Cylinder_Alam_2 OR Rolling_Cylinder_Alam_3 OR Pressure_Fail_1 OR Pressure_Fail_2 OR Pressure_Left_Fail OR Pressure_Right_Fail OR Total_Door_Alam OR Total_Axis_Error OR X4_5 OR Alarm_Pick_Barcode_Fail OR PC_Pause OR Camera1_NG_Pause OR NOT Debug_Model AND ssss AND FPC_up_Unready OR NOT Debug_Model AND ssss AND FPC_down_Unready OR NOT Debug_Model AND ssss AND TRAY_up_Unready OR All_Stop OR NOT Debug_Model AND ssss AND TRAY_down_Unready OR NOT Debug_Model AND ssss AND Feed1_UnReady;
IF _p1 THEN Axis1_Halt := TRUE; Axis2_Halt := TRUE; Axis3_Halt := TRUE; Axis4_Halt := TRUE; Axis5_Halt := TRUE; Axis6_Halt := TRUE; Axis7_Halt := TRUE; Axis8_Halt := TRUE; Axis9_Halt := TRUE; Axis10_Halt := TRUE; Axis12_Halt := TRUE; Axis11_Halt := TRUE; Axis21_Halt := TRUE; Axis22_Halt := TRUE; Axis23_Halt := TRUE; Axis24_Halt := TRUE; Axis25_Halt := TRUE; Total_PauseStatus := TRUE; Total_Pause := TRUE; END_IF;
(* Network 2: 暂停汇总 *)
UPB(CLK := Total_Emergency);
IF UPB.Q THEN Axis1_Halt := TRUE; Axis2_Halt := TRUE; Axis3_Halt := TRUE; Axis4_Halt := TRUE; Axis5_Halt := TRUE; Axis6_Halt := TRUE; Axis7_Halt := TRUE; Axis8_Halt := TRUE; Axis9_Halt := TRUE; Axis11_Halt := TRUE; Axis12_Halt := TRUE; Axis10_Halt := TRUE; END_IF;
(* Network 3 *)
IF Total_Pause THEN Axis1_MoveAbsolute := FALSE; Axis2_MoveAbsolute := FALSE; Axis3_MoveAbsolute := FALSE; Axis4_MoveAbsolute := FALSE; Axis4_1_MoveAbsolute := FALSE; Axis5_1_MoveAbsolute := FALSE; Axis5_MoveAbsolute := FALSE; Axis6_MoveAbsolute := FALSE; Axis7_MoveAbsolute := FALSE; Axis8_MoveAbsolute := FALSE; Axis9_MoveAbsolute := FALSE; Axis11_MoveAbsolute := FALSE; Axis10_MoveAbsolute1 := FALSE; Axis12_MoveAbsolute := FALSE; Axis10_MoveAbsolute := FALSE; Axis21_MoveAbsolute := FALSE; Axis22_MoveAbsolute := FALSE; Axis23_MoveAbsolute := FALSE; Axis24_MoveAbsolute := FALSE; Axis25_MoveAbsolute := FALSE; END_IF;
(* Network 4 *)
IF Total_Pause THEN Axis12_PTF := FALSE; Axis1_PTF := FALSE; Axis2_PTF := FALSE; Axis3_PTF := FALSE; Axis3_PTF_2 := FALSE; Axis4_PTF := FALSE; Axis5_PTF := FALSE; Axis6_PTF := FALSE; Axis6_PTF_2 := FALSE; Axis7_PTF := FALSE; Axis7_PTF_2 := FALSE; Axis8_PTF := FALSE; Axis8_PTF_2 := FALSE; Axis9_PTF := FALSE; Axis9_PTF_2 := FALSE; Axis11_PTF := FALSE; Axis10_PTF := FALSE; Axis21_PTF := TRUE; Axis22_PTF := TRUE; Axis23_PTF := TRUE; Axis24_PTF := TRUE; Axis25_PTF := TRUE; END_IF;
(* Network 5 *)
IF X4_6 OR All_Rset THEN UP_Down_Alam1 := FALSE; UP_Down_Alam2 := FALSE; Right_Cylinder_Alam_1 := FALSE; Right_Cylinder_Alam_2 := FALSE; Left_Cylinder_Alam_1 := FALSE; Left_Cylinder_Alam_2 := FALSE; Rolling_Cylinder_Alam_1 := FALSE; Rolling_Cylinder_Alam_2 := FALSE; Rolling_Cylinder_Alam_3 := FALSE; Pressure_Fail_1 := FALSE; Pressure_Fail_2 := FALSE; Pressure_Left_Fail := FALSE; Pressure_Right_Fail := FALSE; Total_Door_Alam := FALSE; Total_Axis_Error := FALSE; Axis1_Halt := FALSE; Axis2_Halt := FALSE; Axis3_Halt := FALSE; Axis4_Halt := FALSE; Axis5_Halt := FALSE; Axis6_Halt := FALSE; Axis7_Halt := FALSE; Axis8_Halt := FALSE; Axis9_Halt := FALSE; Axis11_Halt := FALSE; Axis12_Halt := FALSE; Camera1_NG_Pause := FALSE; PC_Pause := FALSE; FPC_up_Unready := FALSE; FPC_down_Unready := FALSE; TRAY_up_Unready := FALSE; TRAY_down_Unready := FALSE; Feed1_UnReady := FALSE; Axis10_Halt := FALSE; Axis21_Halt := FALSE; Axis22_Halt := FALSE; Axis23_Halt := FALSE; Axis24_Halt := FALSE; Axis25_Halt := FALSE; END_IF;
(* Network 6 *)
IF X4_6 OR All_Rset THEN Total_PauseStatus := FALSE; END_IF;
Motion_Alam_Rst := X4_6 OR All_Rset;
(* Network 7 *)
IF (X4_4 OR All_Start) AND Total_Pause THEN Total_Pause := FALSE; END_IF;
END_PROGRAM

(* POU Other_Folder/Akam_Stop_Message/Emergency_Stop, LD *)
PROGRAM Emergency_Stop
VAR
	AAAAAA: BOOL;
END_VAR
VAR (* helpers for the ST form of the networks *)
	_p1 : BOOL;
END_VAR
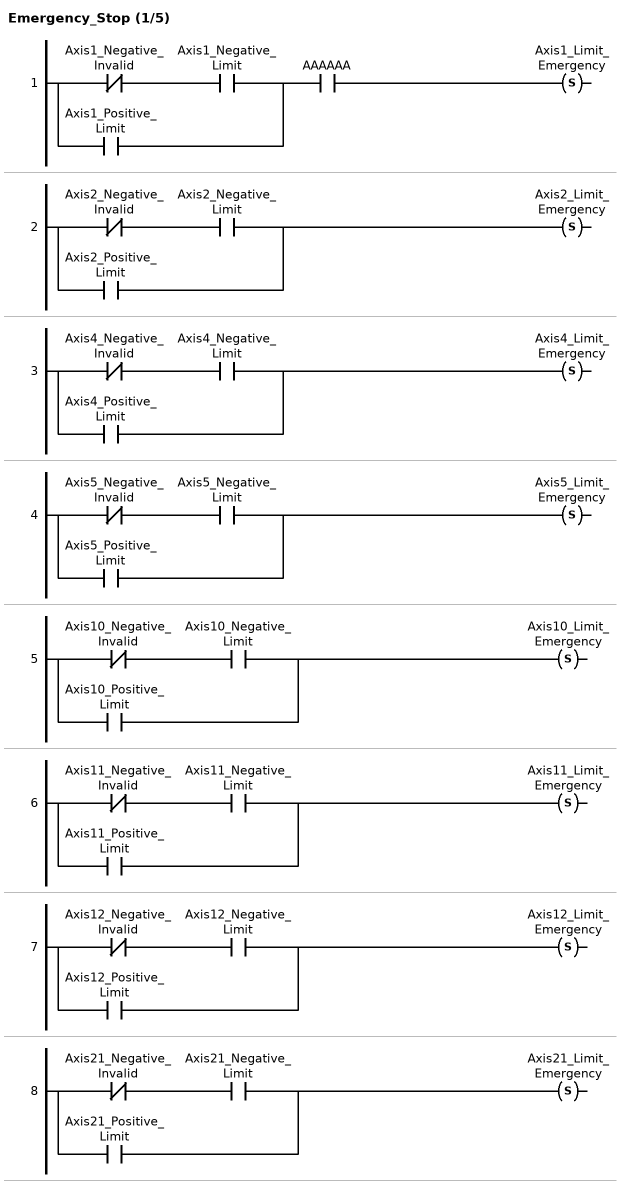
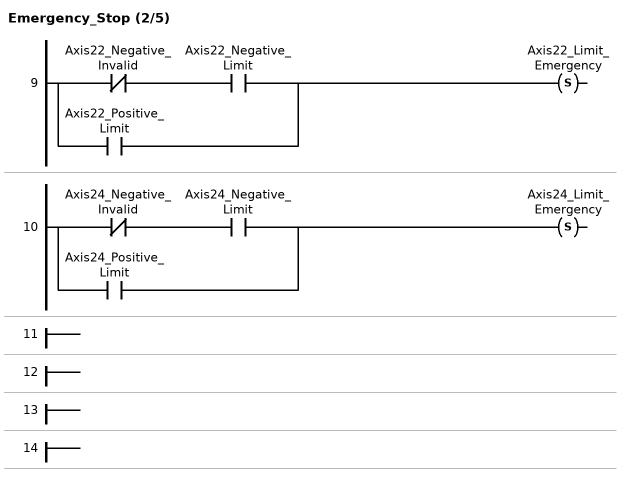
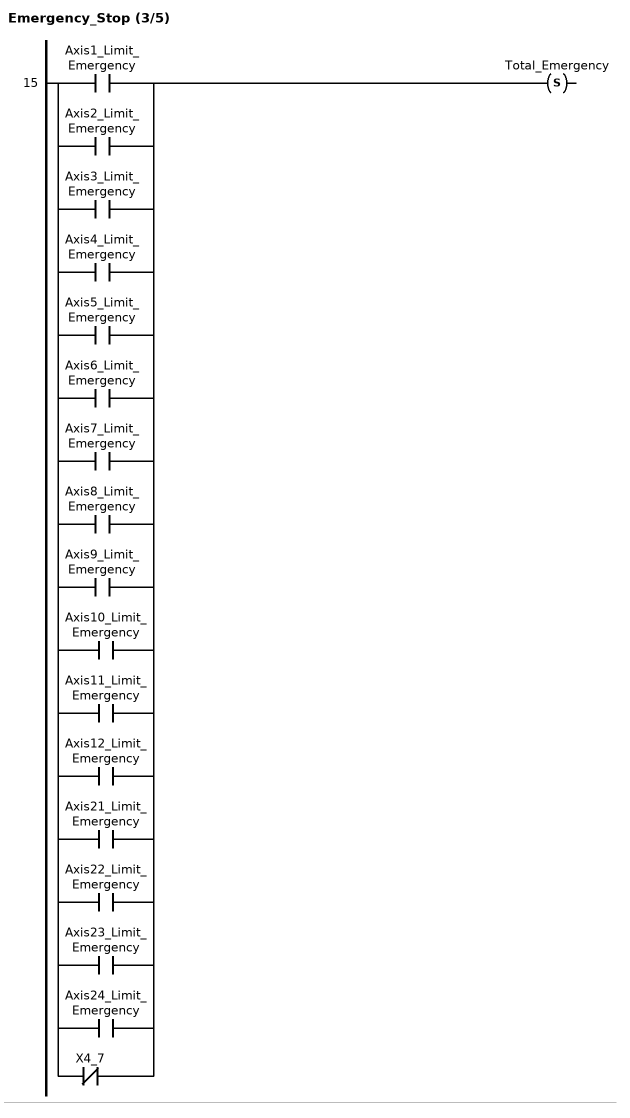
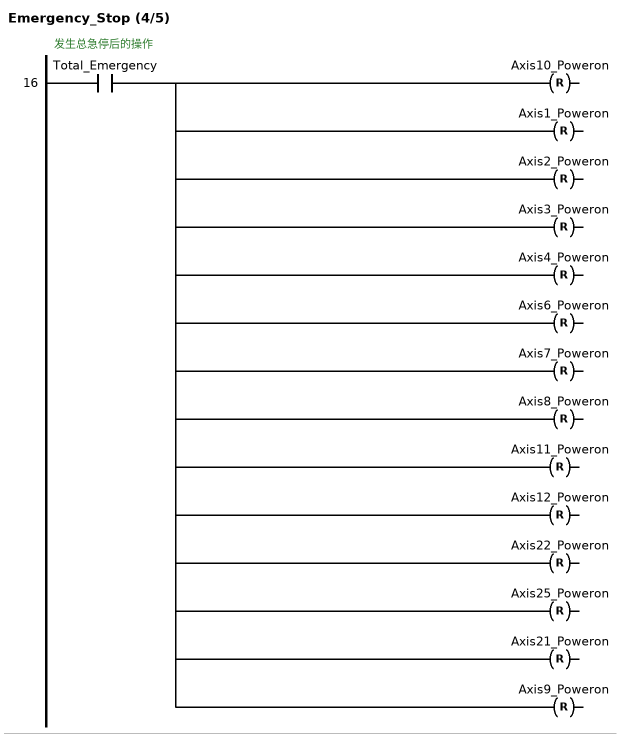
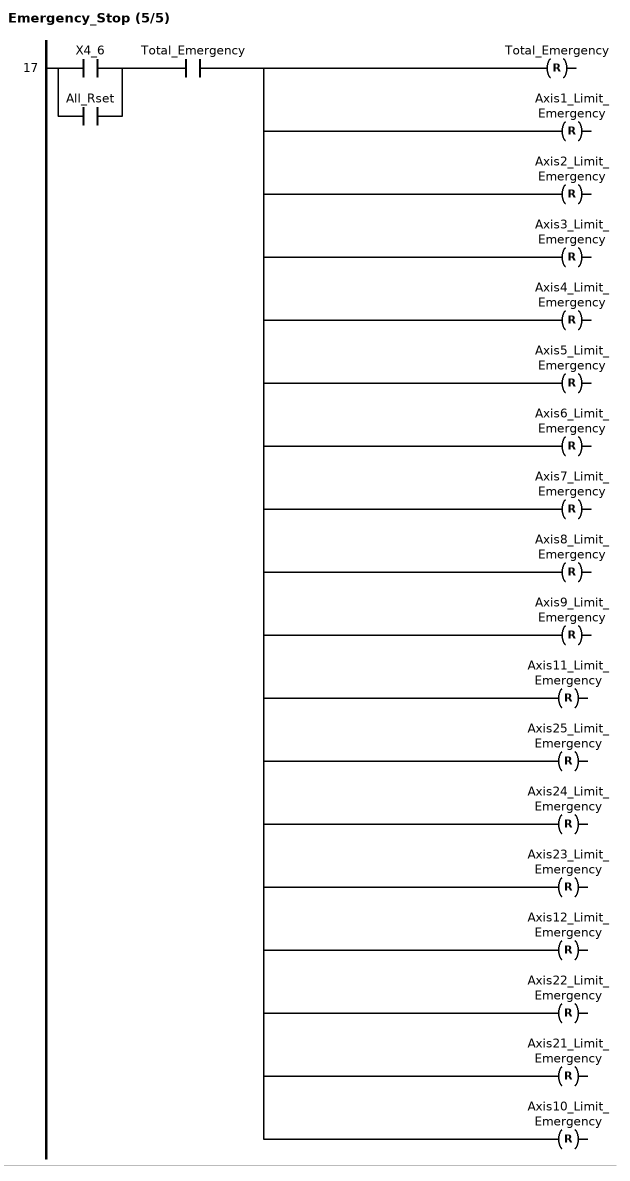
_LD_ (* Ladder Diagram *)
NETWORK 1
	{ [/Axis1_Negative_Invalid] - [Axis1_Negative_Limit] | [Axis1_Positive_Limit] } - [AAAAAA] --- (S Axis1_Limit_Emergency)
NETWORK 2
	{ [/Axis2_Negative_Invalid] - [Axis2_Negative_Limit] | [Axis2_Positive_Limit] } --- (S Axis2_Limit_Emergency)
NETWORK 3
	{ [/Axis4_Negative_Invalid] - [Axis4_Negative_Limit] | [Axis4_Positive_Limit] } --- (S Axis4_Limit_Emergency)
NETWORK 4
	{ [/Axis5_Negative_Invalid] - [Axis5_Negative_Limit] | [Axis5_Positive_Limit] } --- (S Axis5_Limit_Emergency)
NETWORK 5
	{ [/Axis10_Negative_Invalid] - [Axis10_Negative_Limit] | [Axis10_Positive_Limit] } --- (S Axis10_Limit_Emergency)
NETWORK 6
	{ [/Axis11_Negative_Invalid] - [Axis11_Negative_Limit] | [Axis11_Positive_Limit] } --- (S Axis11_Limit_Emergency)
NETWORK 7
	{ [/Axis12_Negative_Invalid] - [Axis12_Negative_Limit] | [Axis12_Positive_Limit] } --- (S Axis12_Limit_Emergency)
NETWORK 8
	{ [/Axis21_Negative_Invalid] - [Axis21_Negative_Limit] | [Axis21_Positive_Limit] } --- (S Axis21_Limit_Emergency)
NETWORK 9
	{ [/Axis22_Negative_Invalid] - [Axis22_Negative_Limit] | [Axis22_Positive_Limit] } --- (S Axis22_Limit_Emergency)
NETWORK 10
	{ [/Axis24_Negative_Invalid] - [Axis24_Negative_Limit] | [Axis24_Positive_Limit] } --- (S Axis24_Limit_Emergency)
NETWORK 11
	*
NETWORK 12
	*
NETWORK 13
	*
NETWORK 14
	*
NETWORK 15
	{ [Axis1_Limit_Emergency] | [Axis2_Limit_Emergency] | [Axis3_Limit_Emergency] | [Axis4_Limit_Emergency] | [Axis5_Limit_Emergency] | [Axis6_Limit_Emergency] | [Axis7_Limit_Emergency] | [Axis8_Limit_Emergency] | [Axis9_Limit_Emergency] | [Axis10_Limit_Emergency] | [Axis11_Limit_Emergency] | [Axis12_Limit_Emergency] | [Axis21_Limit_Emergency] | [Axis22_Limit_Emergency] | [Axis23_Limit_Emergency] | [Axis24_Limit_Emergency] | [/X4_7] } --- (S Total_Emergency)
NETWORK 16 (* 发生总急停后的操作 *)
	[Total_Emergency] --- (R Axis10_Poweron) (R Axis1_Poweron) (R Axis2_Poweron) (R Axis3_Poweron) (R Axis4_Poweron) (R Axis6_Poweron) (R Axis7_Poweron) (R Axis8_Poweron) (R Axis11_Poweron) (R Axis12_Poweron) (R Axis22_Poweron) (R Axis25_Poweron) (R Axis21_Poweron) (R Axis9_Poweron)
NETWORK 17
	{ [X4_6] | [All_Rset] } - [Total_Emergency] --- (R Total_Emergency) (R Axis1_Limit_Emergency) (R Axis2_Limit_Emergency) (R Axis3_Limit_Emergency) (R Axis4_Limit_Emergency) (R Axis5_Limit_Emergency) (R Axis6_Limit_Emergency) (R Axis7_Limit_Emergency) (R Axis8_Limit_Emergency) (R Axis9_Limit_Emergency) (R Axis11_Limit_Emergency) (R Axis25_Limit_Emergency) (R Axis24_Limit_Emergency) (R Axis23_Limit_Emergency) (R Axis12_Limit_Emergency) (R Axis22_Limit_Emergency) (R Axis21_Limit_Emergency) (R Axis10_Limit_Emergency)
_END_LD_
(* the same logic as Structured Text *)
(* Network 1 *)
IF (NOT Axis1_Negative_Invalid AND Axis1_Negative_Limit OR Axis1_Positive_Limit) AND AAAAAA THEN Axis1_Limit_Emergency := TRUE; END_IF;
(* Network 2 *)
IF NOT Axis2_Negative_Invalid AND Axis2_Negative_Limit OR Axis2_Positive_Limit THEN Axis2_Limit_Emergency := TRUE; END_IF;
(* Network 3 *)
IF NOT Axis4_Negative_Invalid AND Axis4_Negative_Limit OR Axis4_Positive_Limit THEN Axis4_Limit_Emergency := TRUE; END_IF;
(* Network 4 *)
IF NOT Axis5_Negative_Invalid AND Axis5_Negative_Limit OR Axis5_Positive_Limit THEN Axis5_Limit_Emergency := TRUE; END_IF;
(* Network 5 *)
IF NOT Axis10_Negative_Invalid AND Axis10_Negative_Limit OR Axis10_Positive_Limit THEN Axis10_Limit_Emergency := TRUE; END_IF;
(* Network 6 *)
IF NOT Axis11_Negative_Invalid AND Axis11_Negative_Limit OR Axis11_Positive_Limit THEN Axis11_Limit_Emergency := TRUE; END_IF;
(* Network 7 *)
IF NOT Axis12_Negative_Invalid AND Axis12_Negative_Limit OR Axis12_Positive_Limit THEN Axis12_Limit_Emergency := TRUE; END_IF;
(* Network 8 *)
IF NOT Axis21_Negative_Invalid AND Axis21_Negative_Limit OR Axis21_Positive_Limit THEN Axis21_Limit_Emergency := TRUE; END_IF;
(* Network 9 *)
IF NOT Axis22_Negative_Invalid AND Axis22_Negative_Limit OR Axis22_Positive_Limit THEN Axis22_Limit_Emergency := TRUE; END_IF;
(* Network 10 *)
IF NOT Axis24_Negative_Invalid AND Axis24_Negative_Limit OR Axis24_Positive_Limit THEN Axis24_Limit_Emergency := TRUE; END_IF;
(* Network 11 *)
(* Network 12 *)
(* Network 13 *)
(* Network 14 *)
(* Network 15 *)
IF Axis1_Limit_Emergency OR Axis2_Limit_Emergency OR Axis3_Limit_Emergency OR Axis4_Limit_Emergency OR Axis5_Limit_Emergency OR Axis6_Limit_Emergency OR Axis7_Limit_Emergency OR Axis8_Limit_Emergency OR Axis9_Limit_Emergency OR Axis10_Limit_Emergency OR Axis11_Limit_Emergency OR Axis12_Limit_Emergency OR Axis21_Limit_Emergency OR Axis22_Limit_Emergency OR Axis23_Limit_Emergency OR Axis24_Limit_Emergency OR NOT X4_7 THEN Total_Emergency := TRUE; END_IF;
(* Network 16: 发生总急停后的操作 *)
IF Total_Emergency THEN Axis10_Poweron := FALSE; Axis1_Poweron := FALSE; Axis2_Poweron := FALSE; Axis3_Poweron := FALSE; Axis4_Poweron := FALSE; Axis6_Poweron := FALSE; Axis7_Poweron := FALSE; Axis8_Poweron := FALSE; Axis11_Poweron := FALSE; Axis12_Poweron := FALSE; Axis22_Poweron := FALSE; Axis25_Poweron := FALSE; Axis21_Poweron := FALSE; Axis9_Poweron := FALSE; END_IF;
(* Network 17 *)
_p1 := (X4_6 OR All_Rset) AND Total_Emergency;
IF _p1 THEN Total_Emergency := FALSE; Axis1_Limit_Emergency := FALSE; Axis2_Limit_Emergency := FALSE; Axis3_Limit_Emergency := FALSE; Axis4_Limit_Emergency := FALSE; Axis5_Limit_Emergency := FALSE; Axis6_Limit_Emergency := FALSE; Axis7_Limit_Emergency := FALSE; Axis8_Limit_Emergency := FALSE; Axis9_Limit_Emergency := FALSE; Axis11_Limit_Emergency := FALSE; Axis25_Limit_Emergency := FALSE; Axis24_Limit_Emergency := FALSE; Axis23_Limit_Emergency := FALSE; Axis12_Limit_Emergency := FALSE; Axis22_Limit_Emergency := FALSE; Axis21_Limit_Emergency := FALSE; Axis10_Limit_Emergency := FALSE; END_IF;
END_PROGRAM

(* POU Other_Folder/Akam_Stop_Message/Lamp, LD *)
PROGRAM Lamp
VAR

	TW1: Twinkle;
	TW2: Twinkle;
	TW3: Twinkle;
	TW4: Twinkle;
	Voice: BOOL;
	UP1: R_TRIG;
	TW5: Twinkle1;
	ssss: BOOL;
END_VAR
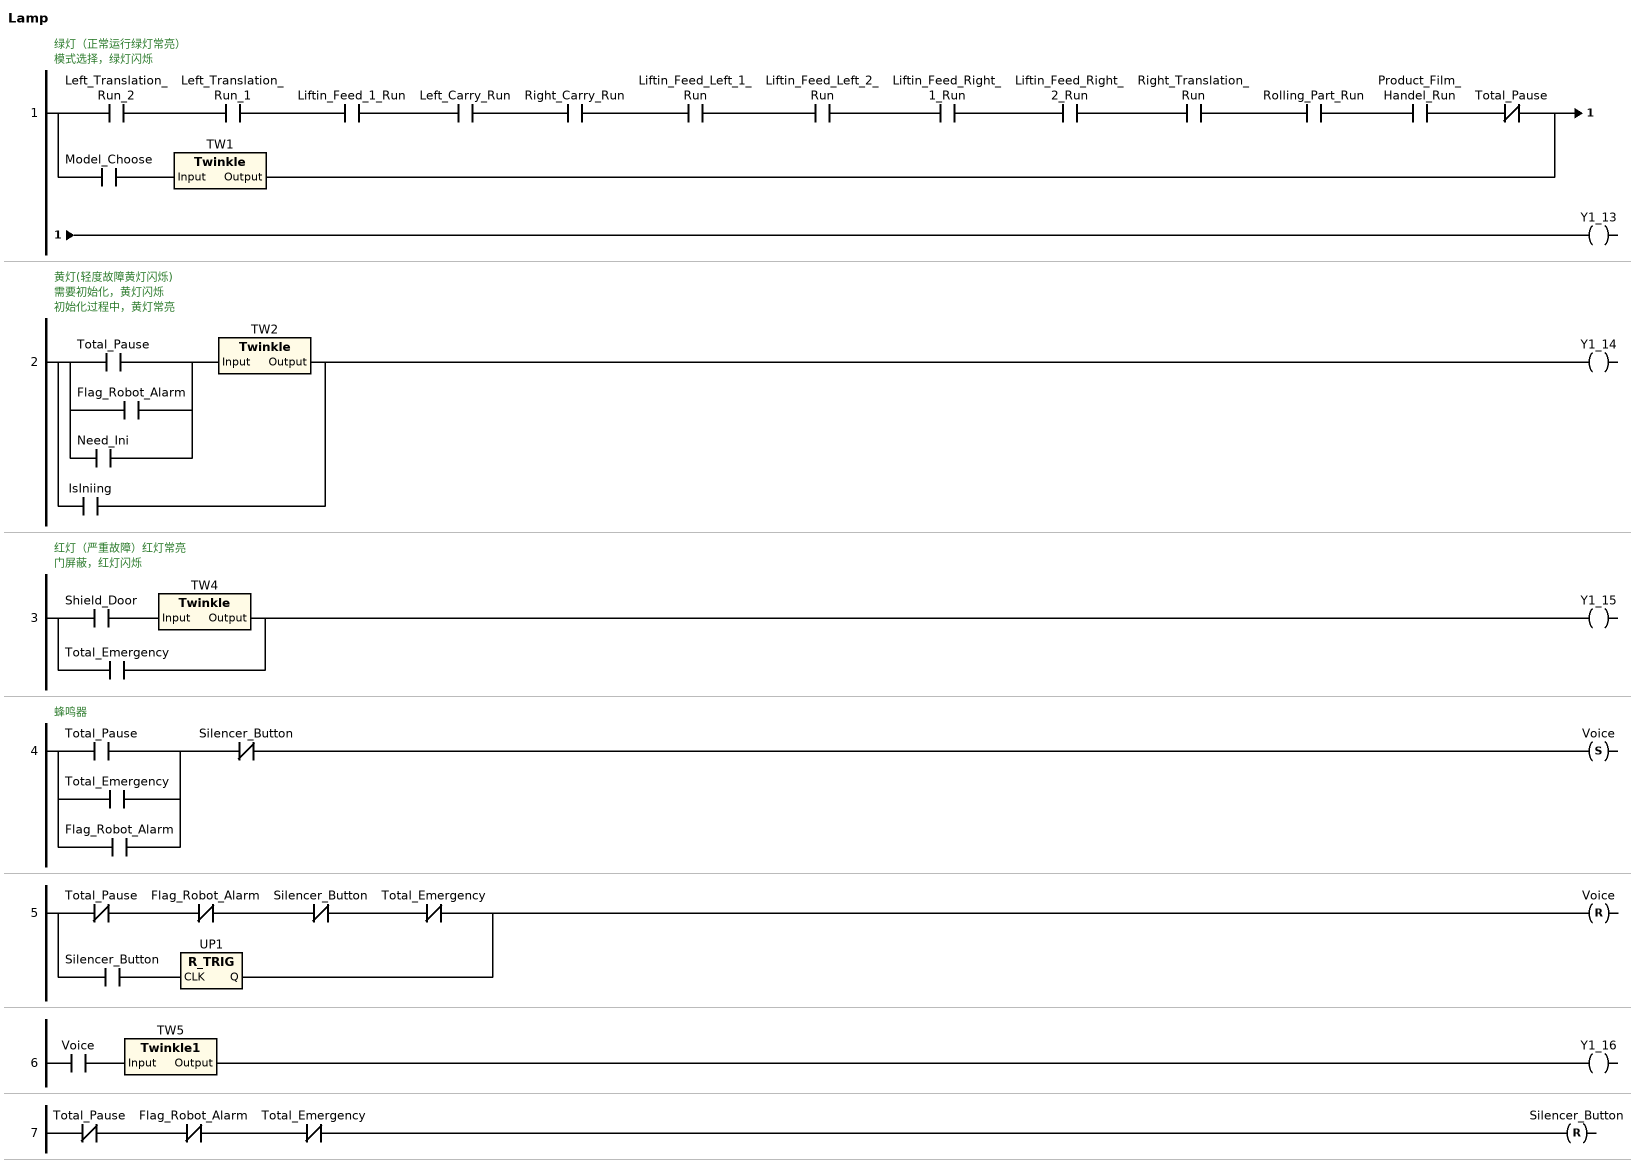
_LD_ (* Ladder Diagram *)
NETWORK 1 (* 绿灯（正常运行绿灯常亮） / 模式选择，绿灯闪烁 *)
	{ [Left_Translation_Run_2] - [Left_Translation_Run_1] - [Liftin_Feed_1_Run] - [Left_Carry_Run] - [Right_Carry_Run] - [Liftin_Feed_Left_1_Run] - [Liftin_Feed_Left_2_Run] - [Liftin_Feed_Right_1_Run] - [Liftin_Feed_Right_2_Run] - [Right_Translation_Run] - [Rolling_Part_Run] - [Product_Film_Handel_Run] - [/Total_Pause] | [Model_Choose] - TW1:Twinkle(Input: *) } --- (Y1_13)
NETWORK 2 (* 黄灯(轻度故障黄灯闪烁) / 需要初始化，黄灯闪烁 / 初始化过程中，黄灯常亮 *)
	{ { [Total_Pause] | [Flag_Robot_Alarm] | [Need_Ini] } - TW2:Twinkle(Input: *) | [IsIniing] } --- (Y1_14)
NETWORK 3 (* 红灯（严重故障）红灯常亮 / 门屏蔽，红灯闪烁 *)
	{ [Shield_Door] - TW4:Twinkle(Input: *) | [Total_Emergency] } --- (Y1_15)
NETWORK 4 (* 蜂鸣器 *)
	{ [Total_Pause] | [Total_Emergency] | [Flag_Robot_Alarm] } - [/Silencer_Button] --- (S Voice)
NETWORK 5
	{ [/Total_Pause] - [/Flag_Robot_Alarm] - [/Silencer_Button] - [/Total_Emergency] | [Silencer_Button] - UP1:R_TRIG(CLK: *) } --- (R Voice)
NETWORK 6
	[Voice] - TW5:Twinkle1(Input: *) --- (Y1_16)
NETWORK 7
	[/Total_Pause] - [/Flag_Robot_Alarm] - [/Total_Emergency] --- (R Silencer_Button)
_END_LD_
(* the same logic as Structured Text *)
(* Network 1: 绿灯（正常运行绿灯常亮） / 模式选择，绿灯闪烁 *)
TW1(Input := Model_Choose);
Y1_13 := Left_Translation_Run_2 AND Left_Translation_Run_1 AND Liftin_Feed_1_Run AND Left_Carry_Run AND Right_Carry_Run AND Liftin_Feed_Left_1_Run AND Liftin_Feed_Left_2_Run AND Liftin_Feed_Right_1_Run AND Liftin_Feed_Right_2_Run AND Right_Translation_Run AND Rolling_Part_Run AND Product_Film_Handel_Run AND NOT Total_Pause OR TW1.Output;
(* Network 2: 黄灯(轻度故障黄灯闪烁) / 需要初始化，黄灯闪烁 / 初始化过程中，黄灯常亮 *)
TW2(Input := Total_Pause OR Flag_Robot_Alarm OR Need_Ini);
Y1_14 := TW2.Output OR IsIniing;
(* Network 3: 红灯（严重故障）红灯常亮 / 门屏蔽，红灯闪烁 *)
TW4(Input := Shield_Door);
Y1_15 := TW4.Output OR Total_Emergency;
(* Network 4: 蜂鸣器 *)
IF (Total_Pause OR Total_Emergency OR Flag_Robot_Alarm) AND NOT Silencer_Button THEN Voice := TRUE; END_IF;
(* Network 5 *)
UP1(CLK := Silencer_Button);
IF NOT Total_Pause AND NOT Flag_Robot_Alarm AND NOT Silencer_Button AND NOT Total_Emergency OR UP1.Q THEN Voice := FALSE; END_IF;
(* Network 6 *)
TW5(Input := Voice);
Y1_16 := TW5.Output;
(* Network 7 *)
IF NOT Total_Pause AND NOT Flag_Robot_Alarm AND NOT Total_Emergency THEN Silencer_Button := FALSE; END_IF;
END_PROGRAM

(* POU Other_Folder/Akam_Stop_Message/Twinkle, LD *)
FUNCTION_BLOCK Twinkle
VAR_INPUT
    Input:BOOL;
END_VAR
VAR_OUTPUT
	Output:BOOL;
END_VAR
VAR
	T0: TON;
	T1: TON;
END_VAR
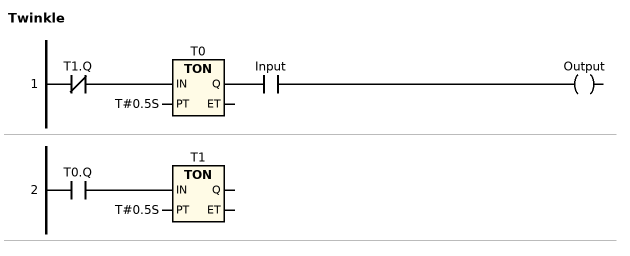
_LD_ (* Ladder Diagram *)
NETWORK 1
	[/T1.Q] - T0:TON(IN: *, PT: T#0.5S) - [Input] --- (Output)
NETWORK 2
	[T0.Q] - T1:TON(IN: *, PT: T#0.5S)
_END_LD_
(* the same logic as Structured Text *)
(* Network 1 *)
T0(IN := NOT T1.Q, PT := T#0.5S);
Output := T0.Q AND Input;
(* Network 2 *)
T1(IN := T0.Q, PT := T#0.5S);
END_FUNCTION_BLOCK

(* POU Other_Folder/Akam_Stop_Message/Twinkle1, LD *)
FUNCTION_BLOCK Twinkle1
VAR_INPUT
    Input:BOOL;
END_VAR
VAR_OUTPUT
	Output:BOOL;
END_VAR
VAR
	T0: TON;
	T1: TON;
END_VAR
